C05396=1037.338,216.569,-106.608,170.716,41.966,157.978
C05397=1037.331,216.320,-106.581,170.714,41.965,157.978
C05398=1037.324,216.072,-106.553,170.711,41.964,157.978
C05399=1037.317,215.823,-106.526,170.708,41.963,157.977
C05400=1037.311,215.576,-106.500,170.706,41.962,157.977
C05401=1037.304,215.327,-106.473,170.703,41.961,157.976
C05402=1037.297,215.079,-106.446,170.701,41.960,157.976
C05403=1037.290,214.829,-106.418,170.698,41.959,157.976
C05404=1037.284,214.582,-106.391,170.696,41.958,157.975
C05405=1037.277,214.333,-106.365,170.693,41.957,157.975
C05406=1037.271,214.084,-106.338,170.691,41.956,157.975
C05407=1037.264,213.837,-106.311,170.689,41.955,157.974
C05408=1037.258,213.587,-106.284,170.686,41.953,157.974
C05409=1037.250,213.339,-106.257,170.684,41.953,157.973
C05410=1037.244,213.091,-106.230,170.681,41.952,157.973
C05411=1037.237,212.842,-106.204,170.679,41.951,157.973
C05412=1037.231,212.593,-106.177,170.676,41.950,157.972
C05413=1037.223,212.345,-106.150,170.674,41.949,157.972
C05414=1037.218,212.097,-106.123,170.672,41.947,157.972
C05415=1037.211,211.848,-106.096,170.670,41.946,157.971
C05416=1037.205,211.600,-106.069,170.668,41.945,157.971
C05417=1037.197,211.351,-106.043,170.665,41.944,157.970
C05418=1037.191,211.102,-106.016,170.663,41.943,157.970
C05419=1037.185,210.854,-105.990,170.660,41.942,157.970
C05420=1037.177,210.606,-105.963,170.658,41.941,157.969
C05421=1037.171,210.357,-105.935,170.656,41.940,157.969
C05422=1037.164,210.109,-105.909,170.653,41.939,157.969
C05423=1037.157,209.860,-105.883,170.651,41.938,157.968
C05424=1037.151,209.611,-105.856,170.648,41.937,157.968
C05425=1037.144,209.364,-105.829,170.646,41.936,157.968
C05426=1037.138,209.115,-105.802,170.644,41.935,157.967
C05427=1037.130,208.866,-105.776,170.641,41.934,157.967
C05428=1037.124,208.618,-105.750,170.639,41.933,157.966
C05429=1037.117,208.369,-105.723,170.636,41.932,157.966
C05430=1037.110,208.120,-105.696,170.634,41.931,157.966
C05431=1037.104,207.872,-105.670,170.632,41.930,157.965
C05432=1037.097,207.623,-105.644,170.629,41.928,157.965
C05433=1037.090,207.376,-105.617,170.627,41.927,157.965
C05434=1037.084,207.127,-105.590,170.624,41.926,157.964
C05435=1037.076,206.878,-105.564,170.622,41.925,157.964
C05436=1037.068,206.555,-105.530,170.619,41.924,157.963
C05437=1037.059,206.231,-105.496,170.616,41.923,157.963
C05438=1037.050,205.907,-105.461,170.613,41.921,157.962
C05439=1037.042,205.583,-105.426,170.610,41.921,157.962
C05440=1037.015,204.533,-105.321,170.301,41.816,157.921
C05441=1037.009,204.284,-105.295,170.298,41.816,157.921
C05442=1037.003,204.035,-105.270,170.295,41.816,157.921
C05443=1036.997,203.787,-105.245,170.292,41.815,157.921
C05444=1036.991,203.537,-105.220,170.288,41.815,157.920
C05445=1036.985,203.289,-105.195,170.285,41.815,157.920
C05446=1036.979,203.041,-105.170,170.282,41.814,157.920
C05447=1036.972,202.792,-105.145,170.279,41.814,157.920
C05448=1036.966,202.543,-105.120,170.275,41.814,157.919
C05449=1036.960,202.295,-105.095,170.272,41.813,157.919
C05450=1036.954,202.046,-105.070,170.269,41.813,157.919
C05451=1036.948,201.797,-105.044,170.266,41.813,157.919
C05452=1036.942,201.549,-105.020,170.262,41.813,157.918
C05453=1036.936,201.300,-104.995,170.259,41.813,157.918
C05454=1036.930,201.051,-104.969,170.256,41.812,157.918
C05455=1036.924,200.802,-104.945,170.253,41.812,157.918
C05456=1036.917,200.554,-104.920,170.250,41.812,157.917
C05457=1036.911,200.305,-104.895,170.246,41.812,157.917
C05458=1036.905,200.057,-104.871,170.243,41.812,157.917
C05459=1036.899,199.808,-104.846,170.241,41.811,157.917
C05460=1036.892,199.559,-104.822,170.238,41.811,157.916
C05461=1036.886,199.310,-104.796,170.234,41.811,157.916
C05462=1036.880,199.061,-104.772,170.231,41.811,157.916
C05463=1036.873,198.813,-104.747,170.228,41.811,157.916
C05464=1036.868,198.564,-104.723,170.225,41.811,157.916
C05465=1036.861,198.316,-104.698,170.222,41.811,157.915
C05466=1036.855,198.066,-104.673,170.219,41.810,157.915
C05467=1036.848,197.818,-104.649,170.215,41.810,157.915
C05468=1036.843,197.570,-104.624,170.212,41.810,157.915
C05469=1036.836,197.321,-104.600,170.209,41.810,157.915
C05470=1036.830,197.072,-104.575,170.206,41.810,157.914
C05471=1036.824,196.823,-104.550,170.203,41.810,157.914
C05472=1036.817,196.575,-104.526,170.199,41.810,157.914
C05473=1036.812,196.326,-104.501,170.196,41.810,157.914
C05474=1036.805,196.077,-104.477,170.193,41.809,157.913
C05475=1036.799,195.828,-104.452,170.190,41.810,157.913
C05476=1036.793,195.580,-104.428,170.187,41.810,157.913
C05477=1036.787,195.331,-104.403,170.184,41.809,157.913
C05478=1036.780,195.082,-104.379,170.180,41.809,157.913
C05479=1036.774,194.833,-104.354,170.177,41.809,157.912
C05480=1036.768,194.585,-104.330,170.174,41.809,157.912
C05481=1036.762,194.336,-104.305,170.172,41.809,157.912
C05482=1036.755,194.087,-104.281,170.169,41.809,157.912
C05483=1036.749,193.839,-104.256,170.165,41.809,157.912
C05484=1036.743,193.590,-104.232,170.162,41.808,157.911
C05485=1036.737,193.341,-104.208,170.159,41.809,157.911
C05486=1036.731,193.092,-104.184,170.156,41.809,157.911
C05487=1036.725,192.844,-104.159,170.153,41.808,157.911
C05488=1036.718,192.595,-104.135,170.150,41.808,157.910
C05489=1036.713,192.346,-104.110,170.147,41.809,157.910
C05490=1036.706,192.097,-104.086,170.144,41.808,157.910
C05491=1036.701,191.849,-104.061,170.141,41.808,157.910
C05492=1036.694,191.600,-104.037,170.138,41.808,157.910
C05493=1036.688,191.351,-104.013,170.135,41.808,157.910
C05494=1036.682,191.103,-103.989,170.132,41.808,157.909
C05495=1036.676,190.853,-103.964,170.128,41.808,157.909
C05496=1036.670,190.606,-103.940,170.125,41.808,157.909
C05497=1036.664,190.356,-103.915,170.122,41.808,157.909
C05498=1036.657,190.107,-103.891,170.120,41.808,157.909
C05499=1036.652,189.859,-103.867,170.117,41.807,157.908
C05500=1036.645,189.610,-103.843,170.114,41.807,157.908
C05501=1036.639,189.326,-103.815,170.110,41.807,157.908
C05502=1036.632,189.041,-103.787,170.106,41.808,157.908
C05503=1036.625,188.758,-103.760,170.103,41.807,157.907
C05504=1036.618,188.473,-103.732,170.100,41.807,157.907
C05505=1036.612,188.225,-103.708,170.097,41.807,157.907
C05506=1036.606,187.976,-103.683,170.094,41.807,157.907
C05507=1036.600,187.728,-103.660,170.091,41.807,157.907
C05508=1036.594,187.478,-103.635,170.088,41.807,157.906
C05509=1036.588,187.230,-103.611,170.085,41.807,157.906
C05510=1036.582,186.981,-103.587,170.082,41.807,157.906
C05511=1036.576,186.732,-103.563,170.079,41.807,157.906
C05512=1036.570,186.483,-103.539,170.075,41.807,157.906
C05513=1036.564,186.235,-103.515,170.073,41.807,157.906
C05514=1036.558,185.986,-103.491,170.070,41.807,157.905
C05515=1036.552,185.737,-103.467,170.067,41.806,157.905
C05516=1036.546,185.488,-103.443,170.064,41.806,157.905
C05517=1036.541,185.239,-103.419,170.062,41.806,157.905
C05518=1036.535,184.991,-103.395,170.059,41.806,157.905
C05519=1036.529,184.742,-103.371,170.055,41.806,157.904
C05520=1036.523,184.493,-103.347,170.052,41.806,157.904
C05521=1036.517,184.244,-103.322,170.049,41.806,157.904
C05522=1036.511,183.996,-103.299,170.047,41.806,157.904
C05523=1036.505,183.746,-103.274,170.044,41.806,157.904
C05524=1036.499,183.498,-103.250,170.041,41.806,157.903
C05525=1036.493,183.250,-103.227,170.037,41.806,157.903
C05526=1036.486,183.000,-103.204,170.035,41.806,157.903
C05527=1036.480,182.752,-103.180,170.032,41.807,157.903
C05528=1036.474,182.503,-103.156,170.029,41.806,157.903
C05529=1036.468,182.254,-103.133,170.026,41.807,157.903
C05530=1036.461,182.005,-103.109,170.023,41.807,157.903
C05531=1036.455,181.757,-103.085,170.020,41.807,157.902
C05532=1036.449,181.507,-103.062,170.018,41.807,157.902
C05533=1036.442,181.259,-103.039,170.015,41.807,157.902
C05534=1036.436,181.010,-103.015,170.012,41.807,157.902
C05535=1036.430,180.761,-102.992,170.009,41.808,157.902
C05536=1036.423,180.512,-102.968,170.005,41.808,157.902
C05537=1036.418,180.264,-102.945,170.002,41.808,157.902
C05538=1036.411,180.015,-102.921,170.000,41.808,157.901
C05539=1036.405,179.766,-102.898,169.997,41.808,157.901
C05540=1036.399,179.517,-102.874,169.994,41.809,157.901
C05541=1036.393,179.268,-102.851,169.991,41.809,157.901
C05542=1036.386,179.020,-102.828,169.988,41.809,157.901
C05543=1036.380,178.770,-102.805,169.986,41.809,157.901
C05544=1036.374,178.522,-102.781,169.983,41.810,157.901
C05545=1036.367,178.272,-102.758,169.979,41.809,157.900
C05546=1036.361,178.024,-102.734,169.976,41.810,157.900
C05547=1036.356,177.775,-102.711,169.974,41.810,157.900
C05548=1036.349,177.526,-102.687,169.971,41.810,157.900
C05549=1036.342,177.278,-102.665,169.968,41.810,157.900
C05550=1036.336,177.029,-102.641,169.965,41.811,157.900
C05551=1036.330,176.780,-102.618,169.963,41.810,157.900
C05552=1036.324,176.531,-102.594,169.960,41.811,157.899
C05553=1036.318,176.282,-102.571,169.957,41.811,157.899
C05554=1036.312,176.033,-102.548,169.954,41.811,157.899
C05555=1036.306,175.785,-102.524,169.952,41.811,157.899
C05556=1036.299,175.535,-102.501,169.949,41.812,157.899
C05557=1036.293,175.287,-102.478,169.946,41.812,157.899
C05558=1036.287,175.038,-102.455,169.942,41.812,157.899
C05559=1036.281,174.789,-102.431,169.940,41.812,157.899
C05560=1036.275,174.540,-102.408,169.937,41.813,157.898
C05561=1036.269,174.291,-102.385,169.934,41.812,157.898
C05562=1036.263,174.043,-102.362,169.931,41.813,157.898
C05563=1036.256,173.794,-102.338,169.929,41.813,157.898
C05564=1036.250,173.545,-102.315,169.926,41.813,157.898
C05565=1036.244,173.261,-102.288,169.923,41.813,157.898
C05566=1036.236,172.976,-102.262,169.920,41.814,157.898
C05567=1036.230,172.692,-102.235,169.916,41.813,157.897
C05568=1036.222,172.406,-102.209,169.913,41.814,157.897
C05569=1036.216,172.158,-102.186,169.910,41.814,157.897
C05570=1036.211,171.909,-102.163,169.907,41.814,157.897
C05571=1036.204,171.661,-102.140,169.904,41.814,157.897
C05572=1036.198,171.411,-102.117,169.902,41.815,157.897
C05573=1036.192,171.162,-102.094,169.899,41.815,157.897
C05574=1036.186,170.914,-102.070,169.896,41.815,157.896
C05575=1036.180,170.665,-102.048,169.894,41.815,157.896
C05576=1036.174,170.415,-102.024,169.891,41.816,157.896
C05577=1036.167,170.167,-102.002,169.888,41.816,157.896
C05578=1036.162,169.918,-101.979,169.886,41.816,157.896
C05579=1036.156,169.670,-101.955,169.883,41.816,157.896
C05580=1036.150,169.421,-101.932,169.879,41.817,157.896
C05581=1036.144,169.171,-101.909,169.877,41.816,157.895
C05582=1036.137,168.923,-101.887,169.874,41.817,157.895
C05583=1036.131,168.674,-101.864,169.871,41.817,157.895
C05584=1036.126,168.425,-101.841,169.869,41.817,157.895
C05585=1036.120,168.176,-101.817,169.866,41.817,157.895
C05586=1036.114,167.928,-101.794,169.863,41.818,157.895
C05587=1036.107,167.679,-101.772,169.861,41.818,157.895
C05588=1036.101,167.429,-101.749,169.858,41.818,157.895
C05589=1036.095,167.180,-101.726,169.856,41.818,157.895
C05590=1036.090,166.932,-101.703,169.853,41.818,157.894
C05591=1036.084,166.683,-101.680,169.850,41.819,157.894
C05592=1036.077,166.434,-101.657,169.847,41.818,157.894
C05593=1036.072,166.185,-101.634,169.844,41.819,157.894
C05594=1036.066,165.936,-101.611,169.841,41.819,157.894
C05595=1036.060,165.687,-101.588,169.839,41.819,157.894
C05596=1036.055,165.439,-101.566,169.836,41.819,157.894
C05597=1036.047,165.189,-101.543,169.834,41.820,157.894
C05598=1036.042,164.940,-101.520,169.831,41.820,157.893
C05599=1036.036,164.691,-101.497,169.828,41.820,157.893
C05600=1036.030,164.443,-101.474,169.826,41.820,157.893
C05601=1036.024,164.194,-101.452,169.823,41.820,157.893
C05602=1036.018,163.945,-101.429,169.821,41.821,157.893
C05603=1036.012,163.696,-101.406,169.818,41.821,157.893
C05604=1036.007,163.447,-101.383,169.814,41.821,157.893
C05605=1036.001,163.198,-101.360,169.812,41.821,157.893
C05606=1035.994,162.950,-101.337,169.809,41.822,157.892
C05607=1035.989,162.701,-101.315,169.807,41.822,157.892
C05608=1035.983,162.452,-101.292,169.804,41.822,157.892
C05609=1035.977,162.203,-101.269,169.801,41.822,157.892
C05610=1035.971,161.955,-101.246,169.799,41.822,157.892
C05611=1035.965,161.706,-101.223,169.796,41.823,157.892
C05612=1035.960,161.456,-101.201,169.794,41.822,157.892
C05613=1035.954,161.207,-101.178,169.791,41.823,157.892
C05614=1035.947,160.959,-101.156,169.789,41.823,157.891
C05615=1035.942,160.710,-101.133,169.786,41.824,157.891
C05616=1035.936,160.461,-101.110,169.784,41.823,157.891
C05617=1035.930,160.212,-101.087,169.780,41.824,157.891
C05618=1035.925,159.962,-101.065,169.777,41.824,157.891
C05619=1035.918,159.714,-101.042,169.775,41.824,157.891
C05620=1035.912,159.465,-101.020,169.772,41.825,157.891
C05621=1035.906,159.216,-100.997,169.770,41.825,157.891
C05622=1035.900,158.967,-100.975,169.767,41.825,157.891
C05623=1035.893,158.719,-100.953,169.764,41.826,157.891
C05624=1035.888,158.470,-100.930,169.762,41.826,157.890
C05625=1035.882,158.220,-100.909,169.759,41.827,157.890
C05626=1035.875,157.972,-100.886,169.757,41.827,157.890
C05627=1035.870,157.722,-100.864,169.754,41.827,157.890
C05628=1035.863,157.474,-100.842,169.751,41.828,157.890
C05629=1035.856,157.189,-100.816,169.748,41.828,157.890
C05630=1035.849,156.904,-100.791,169.745,41.829,157.890
C05631=1035.842,156.618,-100.765,169.743,41.829,157.890
C05632=1035.835,156.333,-100.740,169.740,41.829,157.890
C05633=1035.829,156.085,-100.717,169.737,41.830,157.890
C05634=1035.823,155.835,-100.695,169.734,41.830,157.889
C05635=1035.817,155.587,-100.673,169.732,41.830,157.889
C05636=1035.811,155.337,-100.651,169.729,41.831,157.889
C05637=1035.805,155.088,-100.628,169.727,41.831,157.889
C05638=1035.799,154.839,-100.606,169.724,41.831,157.889
C05639=1035.792,154.591,-100.584,169.722,41.832,157.889
C05640=1035.786,154.342,-100.561,169.719,41.832,157.889
C05641=1035.780,154.093,-100.540,169.717,41.832,157.889
C05642=1035.775,153.844,-100.518,169.714,41.833,157.889
C05643=1035.768,153.596,-100.496,169.711,41.833,157.889
C05644=1035.763,153.346,-100.474,169.709,41.834,157.889
C05645=1035.756,153.097,-100.451,169.706,41.834,157.889
C05646=1035.750,152.848,-100.430,169.704,41.834,157.888
C05647=1035.744,152.600,-100.407,169.700,41.835,157.888
C05648=1035.738,152.350,-100.386,169.698,41.835,157.888
C05649=1035.732,152.101,-100.363,169.695,41.835,157.888
C05650=1035.726,151.852,-100.341,169.692,41.836,157.888
C05651=1035.720,151.603,-100.319,169.690,41.836,157.888
C05652=1035.713,151.355,-100.297,169.687,41.837,157.888
C05653=1035.707,151.105,-100.275,169.685,41.837,157.888
C05654=1035.701,150.857,-100.254,169.682,41.837,157.888
C05655=1035.696,150.608,-100.231,169.680,41.838,157.888
C05656=1035.689,150.359,-100.210,169.677,41.839,157.888
C05657=1035.683,150.109,-100.188,169.675,41.839,157.888
C05658=1035.677,149.861,-100.166,169.672,41.839,157.888
C05659=1035.671,149.612,-100.144,169.670,41.840,157.887
C05660=1035.664,149.362,-100.122,169.667,41.840,157.887
C05661=1035.658,149.114,-100.100,169.665,41.840,157.887
C05662=1035.653,148.865,-100.078,169.662,41.841,157.887
C05663=1035.647,148.616,-100.057,169.660,41.841,157.887
C05664=1035.641,148.367,-100.035,169.657,41.841,157.887
C05665=1035.634,148.118,-100.013,169.655,41.842,157.887
C05666=1035.628,147.869,-99.991,169.652,41.842,157.887
C05667=1035.622,147.620,-99.969,169.650,41.842,157.887
C05668=1035.616,147.371,-99.948,169.647,41.843,157.887
C05669=1035.610,147.122,-99.926,169.644,41.844,157.887
C05670=1035.604,146.873,-99.904,169.642,41.844,157.887
C05671=1035.598,146.624,-99.882,169.639,41.845,157.887
C05672=1035.592,146.375,-99.861,169.637,41.845,157.886
C05673=1035.585,146.126,-99.839,169.634,41.845,157.886
C05674=1035.580,145.877,-99.818,169.632,41.846,157.886
C05675=1035.574,145.628,-99.796,169.629,41.847,157.886
C05676=1035.567,145.379,-99.775,169.627,41.847,157.886
C05677=1035.561,145.130,-99.753,169.624,41.847,157.886
C05678=1035.555,144.881,-99.731,169.622,41.848,157.886
C05679=1035.549,144.632,-99.709,169.619,41.848,157.886
C05680=1035.543,144.383,-99.688,169.617,41.849,157.886
C05681=1035.537,144.134,-99.666,169.614,41.849,157.886
C05682=1035.530,143.885,-99.645,169.612,41.850,157.886
C05683=1035.524,143.636,-99.623,169.609,41.850,157.886
C05684=1035.518,143.388,-99.602,169.607,41.850,157.886
C05685=1035.512,143.138,-99.580,169.604,41.851,157.886
C05686=1035.506,142.889,-99.559,169.602,41.852,157.886
C05687=1035.500,142.640,-99.537,169.599,41.852,157.886
C05688=1035.494,142.391,-99.516,169.597,41.852,157.886
C05689=1035.488,142.142,-99.494,169.594,41.853,157.885
C05690=1035.482,141.893,-99.473,169.592,41.853,157.885
C05691=1035.476,141.644,-99.451,169.589,41.854,157.885
C05692=1035.469,141.395,-99.430,169.587,41.854,157.885
C05693=1035.462,141.110,-99.405,169.584,41.855,157.885
C05694=1035.456,140.824,-99.381,169.581,41.855,157.885
C05695=1035.449,140.539,-99.356,169.578,41.856,157.885
C05696=1035.442,140.254,-99.331,169.576,41.857,157.885
C05697=1035.436,140.005,-99.310,169.573,41.857,157.885
C05698=1035.430,139.755,-99.289,169.571,41.857,157.885
C05699=1035.423,139.506,-99.268,169.568,41.858,157.885
C05700=1035.418,139.258,-99.247,169.566,41.858,157.885
C05701=1035.412,139.009,-99.225,169.563,41.859,157.885
C05702=1035.405,138.759,-99.203,169.561,41.859,157.885
C05703=1035.399,138.510,-99.182,169.558,41.860,157.885
C05704=1035.393,138.262,-99.161,169.556,41.860,157.885
C05705=1035.387,138.012,-99.140,169.553,41.861,157.885
C05706=1035.381,137.763,-99.118,169.551,41.861,157.884
C05707=1035.375,137.515,-99.098,169.548,41.862,157.884
C05708=1035.368,137.266,-99.076,169.546,41.862,157.884
C05709=1035.362,137.016,-99.054,169.543,41.863,157.884
C05710=1035.357,136.767,-99.034,169.541,41.864,157.884
C05711=1035.350,136.518,-99.013,169.539,41.864,157.884
C05712=1035.344,136.269,-98.991,169.536,41.865,157.884
C05713=1035.338,136.021,-98.970,169.534,41.865,157.884
C05714=1035.332,135.771,-98.950,169.531,41.866,157.884
C05715=1035.326,135.522,-98.928,169.529,41.866,157.884
C05716=1035.320,135.273,-98.907,169.526,41.867,157.884
C05717=1035.313,135.025,-98.886,169.524,41.867,157.884
C05718=1035.307,134.775,-98.865,169.521,41.868,157.884
C05719=1035.301,134.527,-98.844,169.520,41.869,157.884
C05720=1035.295,134.277,-98.822,169.516,41.869,157.884
C05721=1035.289,134.027,-98.802,169.514,41.869,157.884
C05722=1035.283,133.779,-98.781,169.513,41.870,157.884
C05723=1035.277,133.530,-98.759,169.510,41.871,157.884
C05724=1035.271,133.280,-98.738,169.508,41.871,157.884
C05725=1035.264,133.032,-98.718,169.505,41.871,157.884
C05726=1035.258,132.783,-98.696,169.503,41.872,157.884
C05727=1035.252,132.534,-98.676,169.500,41.873,157.883
C05728=1035.246,132.285,-98.654,169.498,41.873,157.883
C05729=1035.240,132.035,-98.634,169.496,41.874,157.883
C05730=1035.234,131.787,-98.613,169.493,41.874,157.883
C05731=1035.228,131.538,-98.591,169.491,41.875,157.883
C05732=1035.222,131.289,-98.571,169.488,41.875,157.883
C05733=1035.216,131.040,-98.550,169.486,41.876,157.883
C05734=1035.210,130.790,-98.529,169.483,41.876,157.883
C05735=1035.203,130.542,-98.508,169.481,41.877,157.883
C05736=1035.197,130.292,-98.488,169.478,41.878,157.883
C05737=1035.191,130.044,-98.466,169.476,41.878,157.883
C05738=1035.185,129.794,-98.446,169.474,41.879,157.883
C05739=1035.178,129.545,-98.425,169.471,41.879,157.883
C05740=1035.172,129.296,-98.404,169.469,41.880,157.883
C05741=1035.166,129.047,-98.383,169.466,41.881,157.883
C05742=1035.160,128.798,-98.363,169.464,41.882,157.883
C05743=1035.154,128.549,-98.343,169.461,41.882,157.883
C05744=1035.147,128.300,-98.322,169.459,41.882,157.883
C05745=1035.141,128.051,-98.302,169.456,41.883,157.883
C05746=1035.135,127.802,-98.280,169.454,41.884,157.883
C05747=1035.129,127.553,-98.260,169.451,41.885,157.883
C05748=1035.122,127.303,-98.240,169.449,41.885,157.883
C05749=1035.116,127.055,-98.219,169.448,41.886,157.883
C05750=1035.110,126.805,-98.198,169.445,41.886,157.883
C05751=1035.103,126.556,-98.178,169.442,41.887,157.883
C05752=1035.097,126.308,-98.157,169.440,41.888,157.883
C05753=1035.091,126.058,-98.136,169.438,41.888,157.883
C05754=1035.085,125.809,-98.116,169.435,41.889,157.883
C05755=1035.078,125.560,-98.095,169.433,41.889,157.883
C05756=1035.073,125.311,-98.075,169.431,41.890,157.883
C05757=1035.065,125.026,-98.052,169.428,41.891,157.883
C05758=1035.058,124.740,-98.028,169.425,41.892,157.883
C05759=1035.051,124.454,-98.004,169.422,41.892,157.882
C05760=1035.044,124.169,-97.980,169.420,41.893,157.883
C05761=1035.038,123.920,-97.960,169.417,41.894,157.882
C05762=1035.032,123.670,-97.939,169.415,41.894,157.882
C05763=1035.026,123.421,-97.919,169.412,41.895,157.882
C05764=1035.019,123.173,-97.898,169.410,41.895,157.882
C05765=1035.014,122.923,-97.878,169.407,41.896,157.882
C05766=1035.008,122.675,-97.858,169.405,41.897,157.882
C05767=1035.001,122.425,-97.837,169.403,41.897,157.882
C05768=1034.995,122.177,-97.817,169.400,41.898,157.882
C05769=1034.989,121.927,-97.796,169.398,41.898,157.882
C05770=1034.983,121.678,-97.776,169.397,41.899,157.882
C05771=1034.976,121.429,-97.756,169.393,41.900,157.882
C05772=1034.970,121.180,-97.736,169.392,41.900,157.882
C05773=1034.964,120.931,-97.714,169.389,41.901,157.882
C05774=1034.958,120.682,-97.694,169.387,41.901,157.882
C05775=1034.952,120.432,-97.674,169.385,41.902,157.882
C05776=1034.946,120.183,-97.653,169.382,41.903,157.882
C05777=1034.940,119.935,-97.633,169.380,41.903,157.882
C05778=1034.934,119.685,-97.613,169.377,41.904,157.882
C05779=1034.928,119.436,-97.593,169.375,41.904,157.882
C05780=1034.922,119.187,-97.571,169.373,41.905,157.882
C05781=1034.916,118.938,-97.551,169.370,41.906,157.882
C05782=1034.910,118.689,-97.531,169.368,41.906,157.882
C05783=1034.903,118.440,-97.511,169.366,41.907,157.882
C05784=1034.898,118.191,-97.490,169.363,41.907,157.882
C05785=1034.891,117.941,-97.470,169.361,41.908,157.882
C05786=1034.885,117.692,-97.450,169.359,41.908,157.882
C05787=1034.879,117.444,-97.430,169.356,41.909,157.882
C05788=1034.873,117.194,-97.409,169.354,41.910,157.882
C05789=1034.867,116.945,-97.389,169.351,41.910,157.882
C05790=1034.861,116.697,-97.369,169.349,41.911,157.882
C05791=1034.854,116.447,-97.348,169.347,41.911,157.882
C05792=1034.849,116.198,-97.328,169.344,41.912,157.881
C05793=1034.843,115.949,-97.308,169.342,41.913,157.882
C05794=1034.837,115.700,-97.288,169.340,41.913,157.881
C05795=1034.831,115.451,-97.268,169.338,41.914,157.882
C05796=1034.825,115.202,-97.247,169.335,41.914,157.881
C05797=1034.819,114.952,-97.227,169.333,41.915,157.881
C05798=1034.813,114.704,-97.207,169.331,41.916,157.881
C05799=1034.807,114.455,-97.187,169.329,41.916,157.881
C05800=1034.800,114.205,-97.166,169.327,41.916,157.881
C05801=1034.795,113.956,-97.146,169.324,41.917,157.881
C05802=1034.789,113.707,-97.126,169.322,41.918,157.881
C05803=1034.783,113.457,-97.106,169.320,41.918,157.881
C05804=1034.777,113.208,-97.086,169.317,41.919,157.881
C05805=1034.771,112.959,-97.066,169.315,41.919,157.881
C05806=1034.764,112.710,-97.046,169.313,41.920,157.881
C05807=1034.758,112.461,-97.026,169.310,41.921,157.881
C05808=1034.752,112.212,-97.006,169.308,41.922,157.881
C05809=1034.745,111.963,-96.986,169.306,41.922,157.881
C05810=1034.739,111.714,-96.966,169.303,41.923,157.881
C05811=1034.734,111.465,-96.947,169.301,41.923,157.881
C05812=1034.727,111.215,-96.926,169.299,41.924,157.881
C05813=1034.721,110.966,-96.906,169.296,41.925,157.881
C05814=1034.715,110.717,-96.886,169.294,41.925,157.881
C05815=1034.709,110.468,-96.866,169.291,41.926,157.881
C05816=1034.703,110.218,-96.847,169.289,41.927,157.881
C05817=1034.697,109.970,-96.827,169.287,41.927,157.881
C05818=1034.691,109.721,-96.807,169.285,41.928,157.881
C05819=1034.684,109.471,-96.788,169.283,41.929,157.881
C05820=1034.678,109.222,-96.768,169.281,41.929,157.881
C05821=1034.671,108.936,-96.745,169.278,41.930,157.881
C05822=1034.664,108.651,-96.723,169.275,41.931,157.881
C05823=1034.656,108.365,-96.700,169.272,41.932,157.881
C05824=1034.649,108.079,-96.677,169.270,41.933,157.881
C05825=1034.643,107.830,-96.658,169.267,41.933,157.881
C05826=1034.637,107.581,-96.638,169.265,41.934,157.881
C05827=1034.631,107.333,-96.618,169.263,41.935,157.881
C05828=1034.625,107.083,-96.598,169.260,41.936,157.881
C05829=1034.619,106.834,-96.579,169.259,41.937,157.881
C05830=1034.612,106.585,-96.559,169.256,41.937,157.881
C05831=1034.606,106.336,-96.540,169.254,41.938,157.881
C05832=1034.600,106.086,-96.520,169.252,41.938,157.881
C05833=1034.594,105.837,-96.500,169.250,41.939,157.881
C05834=1034.588,105.588,-96.480,169.247,41.940,157.881
C05835=1034.581,105.340,-96.461,169.245,41.941,157.881
C05836=1034.575,105.089,-96.441,169.243,41.941,157.881
C05837=1034.569,104.841,-96.421,169.240,41.942,157.881
C05838=1034.563,104.592,-96.401,169.238,41.942,157.881
C05839=1034.556,104.343,-96.383,169.236,41.943,157.881
C05840=1034.550,104.094,-96.363,169.233,41.944,157.881
C05841=1034.544,103.844,-96.343,169.231,41.944,157.881
C05842=1034.538,103.595,-96.323,169.229,41.945,157.881
C05843=1034.532,103.345,-96.304,169.226,41.946,157.881
C05844=1034.526,103.097,-96.285,169.224,41.947,157.881
C05845=1034.520,102.848,-96.265,169.222,41.947,157.881
C05846=1034.513,102.598,-96.245,169.220,41.948,157.881
C05847=1034.508,102.349,-96.226,169.218,41.948,157.881
C05848=1034.501,102.100,-96.207,169.216,41.949,157.881
C05849=1034.495,101.851,-96.187,169.213,41.950,157.881
C05850=1034.489,101.602,-96.167,169.211,41.951,157.881
C05851=1034.484,101.352,-96.148,169.209,41.951,157.881
C05852=1034.476,101.103,-96.128,169.206,41.952,157.881
C05853=1034.471,100.854,-96.109,169.204,41.952,157.881
C05854=1034.465,100.605,-96.089,169.202,41.953,157.881
C05855=1034.459,100.355,-96.070,169.199,41.954,157.881
C05856=1034.453,100.107,-96.050,169.197,41.955,157.881
C05857=1034.447,99.858,-96.031,169.195,41.955,157.881
C05858=1034.440,99.607,-96.012,169.192,41.956,157.881
C05859=1034.434,99.359,-95.992,169.190,41.957,157.881
C05860=1034.428,99.109,-95.973,169.188,41.957,157.881
C05861=1034.421,98.860,-95.954,169.186,41.958,157.881
C05862=1034.415,98.612,-95.934,169.184,41.959,157.881
C05863=1034.409,98.362,-95.916,169.182,41.959,157.881
C05864=1034.402,98.113,-95.897,169.179,41.961,157.881
C05865=1034.396,97.864,-95.877,169.177,41.961,157.881
C05866=1034.390,97.615,-95.858,169.175,41.962,157.881
C05867=1034.384,97.365,-95.839,169.172,41.963,157.881
C05868=1034.377,97.117,-95.820,169.170,41.963,157.881
C05869=1034.371,96.867,-95.800,169.168,41.964,157.881
C05870=1034.365,96.618,-95.782,169.165,41.965,157.881
C05871=1034.359,96.369,-95.762,169.163,41.965,157.881
C05872=1034.352,96.120,-95.743,169.161,41.966,157.881
C05873=1034.346,95.870,-95.723,169.159,41.967,157.881
C05874=1034.340,95.621,-95.705,169.157,41.968,157.881
C05875=1034.334,95.372,-95.686,169.155,41.969,157.881
C05876=1034.327,95.123,-95.666,169.152,41.969,157.881
C05877=1034.322,94.874,-95.647,169.150,41.970,157.881
C05878=1034.315,94.625,-95.628,169.148,41.971,157.881
C05879=1034.310,94.375,-95.609,169.145,41.971,157.881
C05880=1034.303,94.127,-95.590,169.143,41.972,157.881
C05881=1034.297,93.877,-95.570,169.141,41.973,157.881
C05882=1034.291,93.628,-95.552,169.138,41.974,157.881
C05883=1034.285,93.379,-95.533,169.136,41.975,157.881
C05884=1034.279,93.129,-95.514,169.134,41.975,157.881
C05885=1034.271,92.844,-95.492,169.132,41.976,157.881
C05886=1034.264,92.557,-95.470,169.129,41.977,157.881
C05887=1034.257,92.272,-95.448,169.127,41.977,157.881
C05888=1034.250,91.986,-95.426,169.124,41.978,157.881
C05889=1034.244,91.737,-95.407,169.122,41.979,157.881
C05890=1034.238,91.488,-95.388,169.119,41.980,157.880
C05891=1034.231,91.239,-95.369,169.117,41.981,157.881
C05892=1034.226,90.990,-95.350,169.115,41.981,157.880
C05893=1034.219,90.741,-95.331,169.112,41.982,157.881
C05894=1034.214,90.491,-95.312,169.110,41.982,157.880
C05895=1034.207,90.242,-95.293,169.108,41.983,157.881
C05896=1034.201,89.993,-95.274,169.106,41.984,157.881
C05897=1034.195,89.743,-95.255,169.103,41.985,157.880
C05898=1034.189,89.494,-95.237,169.102,41.986,157.881
C05899=1034.182,89.245,-95.218,169.100,41.987,157.881
C05900=1034.176,88.996,-95.199,169.097,41.987,157.880
C05901=1034.170,88.747,-95.180,169.095,41.988,157.881
C05902=1034.164,88.497,-95.162,169.093,41.989,157.881
C05903=1034.157,88.248,-95.143,169.090,41.990,157.881
C05904=1034.151,87.999,-95.124,169.088,41.990,157.881
C05905=1034.145,87.750,-95.105,169.086,41.991,157.881
C05906=1034.139,87.501,-95.086,169.083,41.992,157.881
C05907=1034.132,87.252,-95.068,169.081,41.993,157.881
C05908=1034.126,87.002,-95.049,169.079,41.993,157.881
C05909=1034.119,86.753,-95.030,169.077,41.995,157.881
C05910=1034.113,86.504,-95.012,169.075,41.995,157.881
C05911=1034.107,86.255,-94.993,169.073,41.996,157.881
C05912=1034.101,86.005,-94.975,169.070,41.997,157.881
C05913=1034.095,85.756,-94.956,169.068,41.998,157.881
C05914=1034.088,85.507,-94.937,169.066,41.998,157.881
C05915=1034.082,85.258,-94.919,169.063,41.999,157.881
C05916=1034.075,85.009,-94.900,169.061,42.000,157.881
C05917=1034.070,84.759,-94.881,169.059,42.000,157.881
C05918=1034.063,84.510,-94.862,169.056,42.001,157.881
C05919=1034.057,84.261,-94.844,169.055,42.002,157.881
C05920=1034.051,84.011,-94.826,169.053,42.003,157.881
C05921=1034.044,83.762,-94.807,169.050,42.004,157.881
C05922=1034.038,83.513,-94.788,169.048,42.005,157.881
C05923=1034.032,83.263,-94.769,169.046,42.005,157.881
C05924=1034.026,83.014,-94.750,169.043,42.006,157.881
C05925=1034.020,82.766,-94.732,169.041,42.007,157.881
C05926=1034.014,82.516,-94.714,169.039,42.007,157.881
C05927=1034.007,82.267,-94.696,169.036,42.008,157.881
C05928=1034.001,82.018,-94.677,169.034,42.009,157.881
C05929=1033.995,81.769,-94.658,169.032,42.010,157.881
C05930=1033.989,81.519,-94.640,169.029,42.011,157.881
C05931=1033.983,81.270,-94.621,169.028,42.012,157.881
C05932=1033.976,81.020,-94.602,169.026,42.012,157.881
C05933=1033.970,80.771,-94.584,169.024,42.013,157.881
C05934=1033.964,80.522,-94.566,169.021,42.014,157.881
C05935=1033.958,80.273,-94.548,169.019,42.014,157.881
C05936=1033.952,80.024,-94.529,169.017,42.015,157.881
C05937=1033.946,79.775,-94.510,169.014,42.016,157.881
C05938=1033.940,79.525,-94.492,169.012,42.017,157.881
C05939=1033.933,79.276,-94.473,169.010,42.017,157.881
C05940=1033.927,79.027,-94.454,169.007,42.018,157.881
C05941=1033.921,78.778,-94.437,169.005,42.019,157.881
C05942=1033.915,78.529,-94.418,169.004,42.020,157.881
C05943=1033.908,78.279,-94.400,169.002,42.020,157.881
C05944=1033.902,78.030,-94.382,168.999,42.021,157.881
C05945=1033.896,77.781,-94.363,168.997,42.022,157.881
C05946=1033.890,77.531,-94.344,168.995,42.022,157.881
C05947=1033.883,77.282,-94.326,168.992,42.023,157.881
C05948=1033.878,77.033,-94.308,168.990,42.024,157.881
C05949=1033.870,76.747,-94.286,168.987,42.025,157.881
C05950=1033.863,76.462,-94.266,168.985,42.026,157.881
C05951=1033.856,76.175,-94.245,168.982,42.027,157.881
C05952=1033.849,75.889,-94.224,168.979,42.028,157.881
C05953=1033.843,75.640,-94.206,168.978,42.029,157.881
C05954=1033.837,75.390,-94.188,168.976,42.030,157.881
C05955=1033.830,75.142,-94.170,168.973,42.030,157.881
C05956=1033.824,74.893,-94.152,168.971,42.031,157.881
C05957=1033.817,74.644,-94.133,168.969,42.032,157.881
C05958=1033.811,74.394,-94.115,168.966,42.033,157.881
C05959=1033.805,74.145,-94.097,168.964,42.033,157.881
C05960=1033.799,73.895,-94.079,168.962,42.034,157.881
C05961=1033.793,73.647,-94.061,168.959,42.036,157.881
C05962=1033.786,73.397,-94.043,168.957,42.036,157.881
C05963=1033.780,73.148,-94.025,168.956,42.037,157.881
C05964=1033.774,72.898,-94.007,168.953,42.038,157.881
C05965=1033.768,72.650,-93.988,168.951,42.039,157.881
C05966=1033.762,72.400,-93.970,168.949,42.039,157.881
C05967=1033.755,72.151,-93.952,168.946,42.040,157.881
C05968=1033.749,71.901,-93.934,168.944,42.041,157.881
C05969=1033.742,71.652,-93.917,168.942,42.041,157.881
C05970=1033.736,71.403,-93.898,168.939,42.042,157.881
C05971=1033.730,71.154,-93.880,168.937,42.043,157.881
C05972=1033.724,70.904,-93.862,168.936,42.044,157.881
C05973=1033.718,70.655,-93.844,168.934,42.045,157.881
C05974=1033.712,70.406,-93.826,168.931,42.046,157.881
C05975=1033.705,70.157,-93.808,168.929,42.047,157.881
C05976=1033.699,69.907,-93.790,168.927,42.047,157.881
C05977=1033.693,69.657,-93.772,168.924,42.048,157.881
C05978=1033.687,69.409,-93.754,168.922,42.049,157.881
C05979=1033.681,69.159,-93.736,168.920,42.050,157.881
C05980=1033.674,68.910,-93.719,168.917,42.050,157.881
C05981=1033.668,68.661,-93.700,168.915,42.051,157.881
C05982=1033.662,68.412,-93.682,168.914,42.052,157.881
C05983=1033.655,68.162,-93.665,168.911,42.053,157.881
C05984=1033.649,67.913,-93.646,168.909,42.054,157.881
C05985=1033.643,67.663,-93.629,168.907,42.055,157.881
C05986=1033.636,67.415,-93.612,168.904,42.056,157.881
C05987=1033.630,67.165,-93.594,168.902,42.057,157.881
C05988=1033.624,66.916,-93.575,168.900,42.057,157.881
C05989=1033.618,66.667,-93.557,168.897,42.058,157.881
C05990=1033.611,66.417,-93.540,168.895,42.059,157.881
C05991=1033.605,66.168,-93.522,168.893,42.060,157.881
C05992=1033.599,65.919,-93.505,168.890,42.060,157.881
C05993=1033.593,65.670,-93.487,168.889,42.061,157.881
C05994=1033.587,65.420,-93.469,168.887,42.062,157.881
C05995=1033.580,65.171,-93.451,168.884,42.063,157.881
C05996=1033.574,64.921,-93.434,168.882,42.064,157.881
C05997=1033.568,64.672,-93.416,168.880,42.064,157.881
C05998=1033.561,64.423,-93.398,168.877,42.066,157.881
C05999=1033.555,64.174,-93.380,168.875,42.067,157.882
C06000=1033.548,63.924,-93.363,168.873,42.067,157.882
C06001=1033.542,63.675,-93.345,168.870,42.068,157.881
C06002=1033.537,63.426,-93.327,168.869,42.069,157.882
C06003=1033.530,63.176,-93.310,168.867,42.070,157.882
C06004=1033.523,62.927,-93.293,168.864,42.071,157.882
C06005=1033.518,62.678,-93.275,168.862,42.072,157.882
C06006=1033.511,62.428,-93.258,168.859,42.073,157.882
C06007=1033.504,62.179,-93.240,168.857,42.074,157.882
C06008=1033.498,61.929,-93.222,168.855,42.075,157.882
C06009=1033.492,61.680,-93.205,168.853,42.076,157.882
C06010=1033.485,61.431,-93.188,168.851,42.076,157.882
C06011=1033.479,61.181,-93.170,168.849,42.077,157.882
C06012=1033.472,60.933,-93.153,168.846,42.078,157.882
C06013=1033.465,60.647,-93.133,168.844,42.079,157.882
C06014=1033.457,60.360,-93.114,168.841,42.080,157.882
C06015=1033.450,60.074,-93.094,168.838,42.081,157.882
C06016=1033.443,59.789,-93.073,168.835,42.082,157.882
C06017=1033.436,59.539,-93.056,168.834,42.083,157.882
C06018=1033.431,59.290,-93.039,168.832,42.084,157.882
C06019=1033.424,59.041,-93.021,168.829,42.085,157.882
C06020=1033.417,58.791,-93.004,168.827,42.086,157.882
C06021=1033.411,58.542,-92.987,168.824,42.087,157.882
C06022=1033.405,58.293,-92.969,168.822,42.088,157.882
C06023=1033.398,58.043,-92.952,168.820,42.089,157.882
C06024=1033.392,57.794,-92.934,168.817,42.090,157.882
C06025=1033.385,57.545,-92.917,168.816,42.091,157.882
C06026=1033.379,57.296,-92.900,168.814,42.092,157.882
C06027=1033.372,57.047,-92.883,168.811,42.093,157.882
C06028=1033.366,56.796,-92.865,168.809,42.094,157.882
C06029=1033.360,56.547,-92.848,168.807,42.095,157.882
C06030=1033.353,56.298,-92.831,168.804,42.095,157.882
C06031=1033.348,56.049,-92.814,168.802,42.096,157.882
C06032=1033.341,55.800,-92.796,168.799,42.097,157.882
C06033=1033.335,55.551,-92.779,168.798,42.098,157.882
C06034=1033.329,55.301,-92.761,168.796,42.099,157.883
C06035=1033.322,55.051,-92.745,168.793,42.100,157.883
C06036=1033.316,54.802,-92.728,168.791,42.100,157.882
C06037=1033.310,54.553,-92.710,168.789,42.101,157.883
C06038=1033.303,54.304,-92.693,168.786,42.102,157.883
C06039=1033.297,54.054,-92.675,168.784,42.103,157.883
C06040=1033.291,53.805,-92.659,168.782,42.104,157.883
C06041=1033.284,53.555,-92.641,168.779,42.105,157.883
C06042=1033.278,53.307,-92.624,168.778,42.106,157.883
C06043=1033.271,53.057,-92.607,168.776,42.107,157.883
C06044=1033.266,52.808,-92.590,168.773,42.108,157.883
C06045=1033.259,52.558,-92.573,168.771,42.109,157.883
C06046=1033.253,52.309,-92.556,168.769,42.110,157.883
C06047=1033.247,52.060,-92.538,168.766,42.110,157.883
C06048=1033.241,51.810,-92.522,168.764,42.111,157.883
C06049=1033.234,51.561,-92.504,168.761,42.112,157.883
C06050=1033.228,51.312,-92.487,168.760,42.113,157.883
C06051=1033.222,51.062,-92.469,168.758,42.113,157.883
C06052=1033.216,50.813,-92.453,168.755,42.114,157.883
C06053=1033.209,50.564,-92.436,168.753,42.115,157.883
C06054=1033.203,50.315,-92.418,168.751,42.116,157.883
C06055=1033.197,50.064,-92.402,168.748,42.117,157.883
C06056=1033.191,49.816,-92.385,168.746,42.118,157.883
C06057=1033.184,49.566,-92.367,168.744,42.119,157.883
C06058=1033.178,49.317,-92.350,168.741,42.120,157.883
C06059=1033.172,49.068,-92.333,168.740,42.121,157.883
C06060=1033.165,48.819,-92.316,168.738,42.121,157.883
C06061=1033.160,48.569,-92.299,168.735,42.122,157.883
C06062=1033.153,48.319,-92.282,168.733,42.123,157.883
C06063=1033.147,48.071,-92.265,168.731,42.124,157.883
C06064=1033.140,47.821,-92.248,168.728,42.124,157.883
C06065=1033.135,47.572,-92.231,168.726,42.125,157.883
C06066=1033.129,47.322,-92.214,168.724,42.126,157.883
C06067=1033.122,47.073,-92.197,168.721,42.127,157.883
C06068=1033.116,46.824,-92.180,168.719,42.128,157.883
C06069=1033.110,46.574,-92.163,168.718,42.129,157.883
C06070=1033.104,46.325,-92.146,168.715,42.130,157.883
C06071=1033.098,46.076,-92.130,168.713,42.131,157.883
C06072=1033.092,45.826,-92.112,168.711,42.131,157.883
C06073=1033.086,45.577,-92.095,168.708,42.132,157.883
C06074=1033.080,45.328,-92.079,168.706,42.133,157.883
C06075=1033.073,45.078,-92.061,168.704,42.134,157.883
C06076=1033.067,44.829,-92.044,168.701,42.134,157.883
C06077=1033.060,44.543,-92.025,168.699,42.135,157.883
C06078=1033.053,44.257,-92.006,168.696,42.136,157.883
C06079=1033.046,43.970,-91.987,168.694,42.137,157.883
C06080=1033.038,43.684,-91.967,168.692,42.138,157.883
C06081=1033.033,43.434,-91.950,168.689,42.139,157.883
C06082=1033.027,43.185,-91.933,168.687,42.140,157.883
C06083=1033.020,42.935,-91.916,168.685,42.141,157.883
C06084=1033.014,42.687,-91.899,168.682,42.142,157.883
C06085=1033.008,42.437,-91.883,168.680,42.142,157.883
C06086=1033.001,42.187,-91.867,168.677,42.143,157.883
C06087=1032.995,41.938,-91.850,168.675,42.144,157.883
C06088=1032.989,41.689,-91.833,168.674,42.145,157.883
C06089=1032.982,41.440,-91.816,168.671,42.146,157.883
C06090=1032.976,41.190,-91.800,168.669,42.147,157.883
C06091=1032.970,40.940,-91.783,168.666,42.148,157.883
C06092=1032.964,40.692,-91.766,168.664,42.149,157.883
C06093=1032.958,40.442,-91.750,168.662,42.150,157.883
C06094=1032.951,40.192,-91.733,168.659,42.151,157.883
C06095=1032.945,39.943,-91.716,168.657,42.152,157.883
C06096=1032.939,39.694,-91.700,168.656,42.152,157.884
C06097=1032.933,39.445,-91.684,168.653,42.154,157.884
C06098=1032.926,39.195,-91.666,168.651,42.154,157.883
C06099=1032.920,38.946,-91.650,168.648,42.155,157.883
C06100=1032.914,38.697,-91.634,168.646,42.156,157.884
C06101=1032.908,38.446,-91.617,168.644,42.157,157.884
C06102=1032.901,38.198,-91.600,168.641,42.158,157.884
C06103=1032.895,37.948,-91.584,168.639,42.158,157.884
C06104=1032.889,37.698,-91.567,168.637,42.159,157.884
C06105=1032.883,37.449,-91.551,168.635,42.160,157.884
C06106=1032.877,37.200,-91.534,168.633,42.161,157.884
C06107=1032.871,36.951,-91.518,168.630,42.162,157.884
C06108=1032.863,36.701,-91.502,168.628,42.163,157.884
C06109=1032.857,36.452,-91.486,168.625,42.164,157.884
C06110=1032.851,36.203,-91.469,168.623,42.165,157.884
C06111=1032.845,35.952,-91.453,168.621,42.166,157.884
C06112=1032.838,35.704,-91.436,168.618,42.167,157.884
C06113=1032.832,35.455,-91.420,168.617,42.168,157.884
C06114=1032.825,35.205,-91.404,168.614,42.169,157.884
C06115=1032.819,34.955,-91.387,168.612,42.170,157.884
C06116=1032.813,34.706,-91.372,168.610,42.171,157.884
C06117=1032.807,34.457,-91.355,168.607,42.172,157.884
C06118=1032.800,34.207,-91.339,168.605,42.173,157.884
C06119=1032.794,33.958,-91.322,168.602,42.174,157.884
C06120=1032.787,33.709,-91.306,168.601,42.175,157.884
C06121=1032.781,33.460,-91.290,168.598,42.176,157.884
C06122=1032.775,33.210,-91.273,168.596,42.177,157.884
C06123=1032.768,32.961,-91.258,168.594,42.178,157.884
C06124=1032.762,32.711,-91.241,168.591,42.178,157.884
C06125=1032.756,32.462,-91.225,168.589,42.179,157.884
C06126=1032.750,32.213,-91.209,168.586,42.180,157.884
C06127=1032.743,31.963,-91.193,168.584,42.181,157.884
C06128=1032.737,31.714,-91.176,168.583,42.182,157.884
C06129=1032.731,31.464,-91.160,168.580,42.183,157.884
C06130=1032.725,31.215,-91.144,168.578,42.184,157.884
C06131=1032.718,30.965,-91.128,168.575,42.185,157.884
C06132=1032.712,30.716,-91.112,168.573,42.186,157.884
C06133=1032.706,30.466,-91.095,168.570,42.187,157.884
C06134=1032.700,30.217,-91.079,168.568,42.188,157.884
C06135=1032.693,29.968,-91.064,168.566,42.189,157.884
C06136=1032.687,29.719,-91.047,168.564,42.190,157.884
C06137=1032.681,29.469,-91.031,168.562,42.191,157.884
C06138=1032.674,29.220,-91.015,168.559,42.192,157.885
C06139=1032.668,28.970,-90.999,168.557,42.193,157.885
C06140=1032.662,28.721,-90.982,168.555,42.193,157.884
C06141=1032.653,28.345,-90.959,168.551,42.195,157.885
C06142=1032.643,27.969,-90.934,168.547,42.196,157.885
C06143=1032.634,27.594,-90.911,168.545,42.198,157.885
C06144=1032.624,27.219,-90.887,168.541,42.199,157.885
C06145=1032.618,26.970,-90.870,168.538,42.200,157.885
C06146=1032.612,26.720,-90.854,168.536,42.201,157.885
C06147=1032.605,26.470,-90.839,168.534,42.202,157.885
C06148=1032.599,26.221,-90.822,168.531,42.203,157.885
C06149=1032.589,25.811,-90.796,168.528,42.205,157.885
C06150=1032.578,25.401,-90.770,168.524,42.206,157.885
C06151=1032.567,24.992,-90.744,168.520,42.208,157.885
C06152=1032.557,24.582,-90.719,168.516,42.210,157.885
C06153=1032.551,24.333,-90.703,168.513,42.211,157.885
C06154=1032.545,24.084,-90.687,168.512,42.212,157.885
C06155=1032.539,23.835,-90.671,168.510,42.213,157.885
C06156=1032.532,23.584,-90.655,168.507,42.214,157.885
C06157=1032.526,23.335,-90.639,168.505,42.215,157.885
C06158=1032.519,23.086,-90.623,168.502,42.216,157.885
C06159=1032.513,22.837,-90.608,168.500,42.217,157.885
C06160=1032.507,22.587,-90.592,168.497,42.218,157.885
C06161=1032.500,22.338,-90.577,168.495,42.218,157.885
C06162=1032.494,22.089,-90.560,168.493,42.219,157.885
C06163=1032.488,21.839,-90.545,168.491,42.220,157.885
C06164=1032.482,21.590,-90.529,168.488,42.221,157.885
C06165=1032.475,21.340,-90.514,168.486,42.222,157.885
C06166=1032.470,21.091,-90.498,168.483,42.223,157.885
C06167=1032.463,20.841,-90.482,168.481,42.224,157.885
C06168=1032.457,20.592,-90.466,168.479,42.225,157.885
C06169=1032.451,20.342,-90.451,168.477,42.226,157.885
C06170=1032.444,20.092,-90.434,168.475,42.227,157.886
C06171=1032.437,19.843,-90.419,168.472,42.228,157.886
C06172=1032.432,19.593,-90.403,168.470,42.229,157.886
C06173=1032.425,19.344,-90.388,168.467,42.230,157.886
C06174=1032.419,19.095,-90.373,168.465,42.231,157.886
C06175=1032.413,18.845,-90.356,168.462,42.232,157.886
C06176=1032.406,18.596,-90.341,168.460,42.233,157.886
C06177=1032.400,18.347,-90.326,168.458,42.234,157.886
C06178=1032.394,18.097,-90.310,168.456,42.235,157.886
C06179=1032.387,17.848,-90.295,168.453,42.236,157.886
C06180=1032.381,17.599,-90.279,168.451,42.237,157.886
C06181=1032.374,17.349,-90.264,168.448,42.238,157.886
C06182=1032.368,17.100,-90.248,168.446,42.239,157.886
C06183=1032.362,16.850,-90.233,168.443,42.240,157.886
C06184=1032.355,16.601,-90.217,168.442,42.241,157.886
C06185=1032.349,16.351,-90.202,168.439,42.242,157.886
C06186=1032.343,16.102,-90.186,168.437,42.243,157.886
C06187=1032.336,15.852,-90.171,168.434,42.244,157.886
C06188=1032.331,15.602,-90.155,168.432,42.245,157.886
C06189=1032.324,15.353,-90.140,168.429,42.246,157.886
C06190=1032.318,15.104,-90.125,168.427,42.247,157.886
C06191=1032.312,14.854,-90.109,168.425,42.248,157.886
C06192=1032.305,14.605,-90.094,168.423,42.249,157.886
C06193=1032.299,14.356,-90.078,168.420,42.250,157.886
C06194=1032.293,14.106,-90.062,168.418,42.251,157.886
C06195=1032.287,13.857,-90.048,168.415,42.252,157.886
C06196=1032.281,13.608,-90.032,168.413,42.253,157.886
C06197=1032.274,13.358,-90.017,168.410,42.254,157.886
C06198=1032.268,13.108,-90.002,168.409,42.255,157.886
C06199=1032.261,12.859,-89.987,168.406,42.257,157.886
C06200=1032.255,12.610,-89.972,168.404,42.257,157.886
C06201=1032.247,12.324,-89.954,168.401,42.259,157.886
C06202=1032.240,12.039,-89.936,168.398,42.260,157.887
C06203=1032.233,11.754,-89.920,168.396,42.261,157.887
C06204=1032.225,11.469,-89.902,168.393,42.263,157.887
C06205=1032.219,11.219,-89.887,168.391,42.264,157.887
C06206=1032.212,10.970,-89.871,168.388,42.265,157.887
C06207=1032.206,10.720,-89.856,168.385,42.266,157.887
C06208=1032.200,10.471,-89.842,168.383,42.267,157.887
C06209=1032.194,10.222,-89.827,168.380,42.268,157.887
C06210=1032.187,9.973,-89.811,168.379,42.269,157.887
C06211=1032.181,9.723,-89.796,168.376,42.271,157.887
C06212=1032.174,9.474,-89.781,168.374,42.272,157.887
C06213=1032.168,9.224,-89.766,168.371,42.273,157.887
C06214=1032.162,8.974,-89.752,168.369,42.274,157.887
C06215=1032.155,8.725,-89.736,168.366,42.275,157.887
C06216=1032.149,8.476,-89.721,168.365,42.276,157.887
C06217=1032.142,8.226,-89.706,168.362,42.277,157.887
C06218=1032.136,7.977,-89.691,168.359,42.278,157.887
C06219=1032.130,7.727,-89.676,168.357,42.279,157.887
C06220=1032.124,7.478,-89.661,168.354,42.280,157.887
C06221=1032.117,7.229,-89.646,168.352,42.281,157.887
C06222=1032.111,6.979,-89.631,168.349,42.282,157.887
C06223=1032.104,6.729,-89.616,168.348,42.283,157.887
C06224=1032.098,6.480,-89.601,168.345,42.284,157.887
C06225=1032.092,6.231,-89.586,168.343,42.285,157.887
C06226=1032.086,5.981,-89.571,168.340,42.286,157.887
C06227=1032.079,5.731,-89.557,168.337,42.287,157.887
C06228=1032.073,5.482,-89.542,168.335,42.288,157.888
C06229=1032.066,5.233,-89.526,168.332,42.289,157.888
C06230=1032.060,4.983,-89.511,168.331,42.290,157.888
C06231=1032.054,4.734,-89.496,168.328,42.291,157.888
C06232=1032.048,4.484,-89.481,168.326,42.292,157.888
C06233=1032.041,4.235,-89.466,168.323,42.293,157.888
C06234=1032.035,3.985,-89.452,168.321,42.294,157.888
C06235=1032.029,3.736,-89.437,168.318,42.295,157.888
C06236=1032.023,3.486,-89.422,168.316,42.296,157.888
C06237=1032.016,3.237,-89.407,168.314,42.298,157.888
C06238=1032.010,2.987,-89.392,168.311,42.299,157.888
C06239=1032.004,2.737,-89.377,168.309,42.300,157.888
C06240=1031.998,2.488,-89.363,168.306,42.301,157.888
C06241=1031.991,2.239,-89.348,168.304,42.302,157.888
C06242=1031.985,1.989,-89.333,168.301,42.303,157.888
C06243=1031.979,1.740,-89.318,168.299,42.304,157.888
C06244=1031.973,1.491,-89.303,168.297,42.305,157.888
C06245=1031.966,1.241,-89.288,168.295,42.306,157.888
C06246=1031.960,0.991,-89.273,168.292,42.307,157.888
C06247=1031.954,0.742,-89.259,168.289,42.308,157.888
C06248=1031.948,0.493,-89.244,168.287,42.309,157.888
C06249=1031.942,0.243,-89.229,168.284,42.310,157.888
C06250=1031.935,-0.007,-89.214,168.282,42.311,157.888
C06251=1031.929,-0.256,-89.199,168.280,42.312,157.888
C06252=1031.923,-0.505,-89.184,168.278,42.313,157.888
C06253=1031.917,-0.756,-89.170,168.275,42.314,157.888
C06254=1031.911,-1.005,-89.156,168.272,42.315,157.888
C06255=1031.905,-1.254,-89.141,168.270,42.316,157.888
C06256=1031.898,-1.504,-89.126,168.267,42.317,157.888
C06257=1031.893,-1.753,-89.111,168.266,42.318,157.888
C06258=1031.886,-2.002,-89.096,168.263,42.319,157.888
C06259=1031.880,-2.252,-89.081,168.261,42.320,157.888
C06260=1031.874,-2.501,-89.067,168.258,42.322,157.888
C06261=1031.868,-2.751,-89.052,168.256,42.323,157.889
C06262=1031.862,-3.001,-89.037,168.253,42.324,157.889
C06263=1031.856,-3.250,-89.023,168.250,42.325,157.889
C06264=1031.849,-3.500,-89.008,168.249,42.326,157.889
C06265=1031.842,-3.783,-88.992,168.246,42.327,157.889
C06266=1031.835,-4.066,-88.974,168.243,42.328,157.889
C06267=1031.828,-4.348,-88.959,168.240,42.329,157.889
C06268=1031.821,-4.632,-88.943,168.237,42.331,157.889
C06269=1031.814,-4.882,-88.928,168.234,42.332,157.889
C06270=1031.808,-5.131,-88.913,168.233,42.333,157.889
C06271=1031.802,-5.380,-88.900,168.230,42.334,157.889
C06272=1031.795,-5.630,-88.885,168.227,42.335,157.889
C06273=1031.788,-5.879,-88.870,168.225,42.336,157.889
C06274=1031.783,-6.129,-88.856,168.222,42.337,157.889
C06275=1031.776,-6.379,-88.841,168.220,42.339,157.889
C06276=1031.769,-6.629,-88.828,168.218,42.340,157.889
C06277=1031.764,-6.878,-88.813,168.215,42.341,157.889
C06278=1031.757,-7.127,-88.798,168.213,42.342,157.889
C06279=1031.751,-7.377,-88.785,168.210,42.343,157.889
C06280=1031.745,-7.626,-88.770,168.207,42.344,157.889
C06281=1031.738,-7.876,-88.756,168.205,42.345,157.889
C06282=1031.732,-8.125,-88.742,168.202,42.346,157.889
C06283=1031.726,-8.375,-88.727,168.200,42.348,157.889
C06284=1031.720,-8.624,-88.714,168.198,42.349,157.889
C06285=1031.713,-8.874,-88.699,168.195,42.350,157.889
C06286=1031.706,-9.124,-88.685,168.192,42.351,157.889
C06287=1031.701,-9.373,-88.670,168.190,42.352,157.889
C06288=1031.694,-9.622,-88.656,168.187,42.353,157.890
C06289=1031.688,-9.871,-88.642,168.186,42.354,157.890
C06290=1031.682,-10.121,-88.627,168.183,42.355,157.890
C06291=1031.676,-10.371,-88.613,168.180,42.357,157.890
C06292=1031.669,-10.620,-88.599,168.178,42.358,157.890
C06293=1031.663,-10.870,-88.585,168.175,42.359,157.890
C06294=1031.656,-11.119,-88.571,168.173,42.360,157.890
C06295=1031.650,-11.369,-88.557,168.171,42.361,157.890
C06296=1031.644,-11.618,-88.542,168.168,42.362,157.890
C06297=1031.638,-11.868,-88.528,168.165,42.364,157.890
C06298=1031.632,-12.117,-88.514,168.163,42.365,157.890
C06299=1031.625,-12.367,-88.500,168.160,42.366,157.890
C06300=1031.620,-12.617,-88.486,168.157,42.367,157.890
C06301=1031.612,-12.866,-88.472,168.156,42.368,157.890
C06302=1031.607,-13.116,-88.458,168.153,42.369,157.890
C06303=1031.601,-13.365,-88.443,168.150,42.371,157.890
C06304=1031.594,-13.615,-88.430,168.148,42.372,157.890
C06305=1031.588,-13.864,-88.415,168.145,42.373,157.890
C06306=1031.582,-14.113,-88.402,168.142,42.374,157.890
C06307=1031.576,-14.364,-88.387,168.141,42.375,157.890
C06308=1031.570,-14.613,-88.373,168.138,42.376,157.890
C06309=1031.563,-14.863,-88.359,168.136,42.377,157.890
C06310=1031.557,-15.112,-88.345,168.133,42.378,157.890
C06311=1031.551,-15.362,-88.331,168.130,42.379,157.890
C06312=1031.545,-15.611,-88.317,168.128,42.380,157.890
C06313=1031.538,-15.860,-88.303,168.125,42.381,157.890
C06314=1031.532,-16.110,-88.289,168.123,42.383,157.891
C06315=1031.526,-16.360,-88.275,168.120,42.384,157.891
C06316=1031.519,-16.609,-88.262,168.118,42.385,157.891
C06317=1031.513,-16.859,-88.247,168.115,42.386,157.891
C06318=1031.507,-17.108,-88.234,168.113,42.388,157.891
C06319=1031.501,-17.357,-88.221,168.111,42.389,157.891
C06320=1031.495,-17.608,-88.206,168.108,42.390,157.891
C06321=1031.488,-17.856,-88.192,168.105,42.391,157.891
C06322=1031.481,-18.106,-88.179,168.102,42.392,157.891
C06323=1031.475,-18.356,-88.165,168.100,42.394,157.891
C06324=1031.469,-18.606,-88.151,168.098,42.395,157.891
C06325=1031.463,-18.855,-88.138,168.095,42.396,157.891
C06326=1031.456,-19.105,-88.124,168.093,42.397,157.891
C06327=1031.450,-19.354,-88.110,168.090,42.398,157.891
C06328=1031.444,-19.603,-88.096,168.087,42.400,157.891
C06329=1031.437,-19.886,-88.081,168.084,42.401,157.891
C06330=1031.430,-20.167,-88.065,168.082,42.402,157.891
C06331=1031.423,-20.448,-88.050,168.079,42.404,157.891
C06332=1031.416,-20.730,-88.035,168.076,42.405,157.891
C06333=1031.409,-20.980,-88.021,168.073,42.406,157.891
C06334=1031.403,-21.229,-88.008,168.070,42.407,157.891
C06335=1031.396,-21.478,-87.993,168.069,42.409,157.892
C06336=1031.391,-21.728,-87.979,168.066,42.410,157.892
C06337=1031.384,-21.977,-87.966,168.063,42.411,157.892
C06338=1031.378,-22.227,-87.953,168.061,42.412,157.892
C06339=1031.372,-22.477,-87.939,168.058,42.413,157.892
C06340=1031.366,-22.726,-87.925,168.055,42.414,157.892
C06341=1031.359,-22.976,-87.912,168.053,42.416,157.892
C06342=1031.354,-23.226,-87.898,168.051,42.417,157.892
C06343=1031.347,-23.475,-87.885,168.048,42.418,157.892
C06344=1031.341,-23.725,-87.871,168.045,42.419,157.892
C06345=1031.334,-23.974,-87.858,168.042,42.421,157.892
C06346=1031.329,-24.224,-87.844,168.040,42.422,157.892
C06347=1031.322,-24.474,-87.830,168.038,42.423,157.892
C06348=1031.316,-24.723,-87.817,168.035,42.424,157.892
C06349=1031.310,-24.972,-87.803,168.033,42.425,157.892
C06350=1031.304,-25.222,-87.789,168.030,42.427,157.892
C06351=1031.297,-25.472,-87.776,168.027,42.428,157.892
C06352=1031.291,-25.721,-87.763,168.024,42.429,157.892
C06353=1031.286,-25.970,-87.749,168.023,42.430,157.892
C06354=1031.279,-26.220,-87.735,168.020,42.432,157.892
C06355=1031.273,-26.470,-87.722,168.017,42.433,157.892
C06356=1031.266,-26.719,-87.709,168.014,42.434,157.892
C06357=1031.261,-26.969,-87.695,168.012,42.435,157.892
C06358=1031.254,-27.218,-87.681,168.009,42.436,157.892
C06359=1031.248,-27.468,-87.668,168.007,42.438,157.892
C06360=1031.242,-27.717,-87.655,168.004,42.439,157.892
C06361=1031.235,-27.967,-87.641,168.002,42.440,157.893
C06362=1031.229,-28.217,-87.629,167.999,42.442,157.893
C06363=1031.223,-28.466,-87.615,167.997,42.443,157.893
C06364=1031.217,-28.715,-87.602,167.994,42.444,157.893
C06365=1031.210,-28.965,-87.589,167.991,42.445,157.893
C06366=1031.203,-29.215,-87.575,167.989,42.447,157.893
C06367=1031.198,-29.465,-87.563,167.986,42.448,157.893
C06368=1031.191,-29.714,-87.549,167.983,42.449,157.893
C06369=1031.185,-29.964,-87.536,167.981,42.451,157.893
C06370=1031.178,-30.213,-87.523,167.978,42.452,157.893
C06371=1031.172,-30.463,-87.510,167.976,42.453,157.893
C06372=1031.166,-30.712,-87.497,167.973,42.454,157.893
C06373=1031.159,-30.962,-87.483,167.970,42.456,157.893
C06374=1031.153,-31.211,-87.470,167.968,42.457,157.893
C06375=1031.147,-31.461,-87.457,167.965,42.458,157.893
C06376=1031.141,-31.711,-87.444,167.963,42.459,157.893
C06377=1031.135,-31.960,-87.431,167.960,42.461,157.893
C06378=1031.129,-32.209,-87.417,167.957,42.462,157.893
C06379=1031.122,-32.460,-87.404,167.955,42.464,157.894
C06380=1031.116,-32.709,-87.391,167.952,42.465,157.894
C06381=1031.110,-32.958,-87.378,167.950,42.466,157.894
C06382=1031.104,-33.208,-87.365,167.947,42.467,157.894
C06383=1031.098,-33.457,-87.352,167.944,42.469,157.894
C06384=1031.091,-33.707,-87.339,167.942,42.470,157.894
C06385=1031.085,-33.957,-87.326,167.939,42.471,157.894
C06386=1031.079,-34.206,-87.313,167.937,42.472,157.894
C06387=1031.072,-34.456,-87.299,167.934,42.474,157.894
C06388=1031.066,-34.706,-87.287,167.931,42.475,157.894
C06389=1031.060,-34.955,-87.274,167.928,42.476,157.894
C06390=1031.054,-35.205,-87.261,167.926,42.478,157.894
C06391=1031.048,-35.454,-87.248,167.924,42.479,157.894
C06392=1031.041,-35.704,-87.234,167.921,42.480,157.894
C06393=1031.035,-35.985,-87.220,167.918,42.481,157.894
C06394=1031.029,-36.266,-87.205,167.915,42.483,157.894
C06395=1031.022,-36.546,-87.191,167.912,42.484,157.894
C06396=1031.014,-36.827,-87.176,167.909,42.486,157.894
C06397=1031.008,-37.076,-87.163,167.906,42.487,157.894
C06398=1031.002,-37.326,-87.150,167.903,42.488,157.894
C06399=1030.996,-37.576,-87.137,167.901,42.489,157.894
C06400=1030.990,-37.825,-87.125,167.899,42.491,157.895
C06401=1030.984,-38.075,-87.111,167.896,42.492,157.895
C06402=1030.977,-38.324,-87.098,167.893,42.493,157.895
C06403=1030.972,-38.574,-87.085,167.890,42.494,157.895
C06404=1030.965,-38.823,-87.072,167.889,42.496,157.895
C06405=1030.959,-39.073,-87.060,167.886,42.497,157.895
C06406=1030.953,-39.323,-87.048,167.883,42.498,157.895
C06407=1030.947,-39.572,-87.034,167.880,42.500,157.895
C06408=1030.941,-39.822,-87.022,167.877,42.501,157.895
C06409=1030.934,-40.071,-87.009,167.875,42.503,157.895
C06410=1030.927,-40.321,-86.996,167.872,42.504,157.895
C06411=1030.921,-40.571,-86.984,167.869,42.505,157.895
C06412=1030.914,-40.820,-86.971,167.867,42.507,157.895
C06413=1030.908,-41.070,-86.958,167.864,42.508,157.895
C06414=1030.903,-41.320,-86.946,167.862,42.509,157.895
C06415=1030.896,-41.569,-86.933,167.859,42.511,157.895
C06416=1030.890,-41.819,-86.921,167.856,42.512,157.895
C06417=1030.884,-42.069,-86.908,167.853,42.514,157.895
C06418=1030.878,-42.318,-86.895,167.850,42.515,157.895
C06419=1030.871,-42.567,-86.883,167.848,42.516,157.896
C06420=1030.865,-42.817,-86.870,167.846,42.517,157.896
C06421=1030.859,-43.067,-86.857,167.843,42.519,157.896
C06422=1030.853,-43.316,-86.845,167.840,42.520,157.896
C06423=1030.846,-43.566,-86.833,167.837,42.521,157.896
C06424=1030.840,-43.816,-86.820,167.835,42.523,157.896
C06425=1030.834,-44.065,-86.807,167.832,42.524,157.896
C06426=1030.827,-44.315,-86.795,167.829,42.526,157.896
C06427=1030.822,-44.565,-86.782,167.826,42.527,157.896
C06428=1030.816,-44.814,-86.770,167.825,42.528,157.896
C06429=1030.809,-45.063,-86.757,167.822,42.530,157.896
C06430=1030.803,-45.313,-86.745,167.819,42.531,157.896
C06431=1030.797,-45.563,-86.732,167.816,42.532,157.896
C06432=1030.791,-45.812,-86.720,167.813,42.534,157.896
C06433=1030.785,-46.062,-86.708,167.811,42.535,157.896
C06434=1030.779,-46.311,-86.694,167.808,42.536,157.896
C06435=1030.772,-46.561,-86.683,167.805,42.538,157.897
C06436=1030.766,-46.811,-86.670,167.802,42.539,157.897
C06437=1030.760,-47.061,-86.657,167.801,42.541,157.897
C06438=1030.754,-47.310,-86.645,167.798,42.542,157.897
C06439=1030.748,-47.560,-86.633,167.795,42.543,157.897
C06440=1030.742,-47.809,-86.621,167.792,42.545,157.897
C06441=1030.735,-48.058,-86.608,167.789,42.546,157.897
C06442=1030.730,-48.308,-86.595,167.786,42.547,157.897
C06443=1030.724,-48.558,-86.583,167.784,42.549,157.897
C06444=1030.717,-48.808,-86.571,167.781,42.550,157.897
C06445=1030.711,-49.057,-86.558,167.778,42.551,157.897
C06446=1030.705,-49.307,-86.546,167.776,42.553,157.897
C06447=1030.699,-49.556,-86.534,167.773,42.554,157.897
C06448=1030.693,-49.806,-86.522,167.771,42.555,157.897
C06449=1030.687,-50.056,-86.509,167.768,42.557,157.897
C06450=1030.681,-50.306,-86.497,167.765,42.558,157.897
C06451=1030.675,-50.555,-86.485,167.762,42.560,157.897
C06452=1030.669,-50.805,-86.472,167.760,42.561,157.897
C06453=1030.662,-51.055,-86.460,167.757,42.563,157.898
C06454=1030.656,-51.304,-86.448,167.754,42.564,157.898
C06455=1030.649,-51.553,-86.437,167.751,42.566,157.898
C06456=1030.644,-51.803,-86.424,167.749,42.568,157.898
C06457=1030.636,-52.085,-86.411,167.746,42.569,157.898
C06458=1030.629,-52.366,-86.397,167.742,42.571,157.898
C06459=1030.622,-52.647,-86.384,167.739,42.573,157.898
C06460=1030.614,-52.928,-86.370,167.737,42.574,157.898
C06461=1030.609,-53.178,-86.359,167.734,42.576,157.898
C06462=1030.603,-53.427,-86.346,167.731,42.577,157.898
C06463=1030.596,-53.677,-86.334,167.729,42.579,157.898
C06464=1030.590,-53.927,-86.322,167.726,42.580,157.898
C06465=1030.583,-54.176,-86.310,167.723,42.582,157.899
C06466=1030.578,-54.425,-86.298,167.720,42.583,157.899
C06467=1030.571,-54.676,-86.287,167.717,42.585,157.899
C06468=1030.565,-54.925,-86.275,167.715,42.587,157.899
C06469=1030.559,-55.175,-86.262,167.712,42.588,157.899
C06470=1030.552,-55.425,-86.250,167.709,42.590,157.899
C06471=1030.546,-55.673,-86.239,167.706,42.591,157.899
C06472=1030.540,-55.924,-86.228,167.704,42.593,157.899
C06473=1030.534,-56.173,-86.215,167.701,42.594,157.899
C06474=1030.527,-56.423,-86.203,167.698,42.596,157.899
C06475=1030.521,-56.672,-86.192,167.695,42.598,157.899
C06476=1030.515,-56.922,-86.180,167.693,42.599,157.899
C06477=1030.509,-57.172,-86.168,167.690,42.600,157.899
C06478=1030.502,-57.422,-86.156,167.687,42.602,157.899
C06479=1030.496,-57.671,-86.145,167.684,42.603,157.900
C06480=1030.490,-57.921,-86.133,167.682,42.605,157.900
C06481=1030.484,-58.171,-86.120,167.679,42.606,157.900
C06482=1030.478,-58.420,-86.109,167.676,42.608,157.900
C06483=1030.471,-58.670,-86.098,167.673,42.609,157.900
C06484=1030.465,-58.919,-86.086,167.671,42.611,157.900
C06485=1030.460,-59.169,-86.074,167.668,42.612,157.900
C06486=1030.453,-59.419,-86.062,167.665,42.614,157.900
C06487=1030.447,-59.668,-86.050,167.662,42.616,157.900
C06488=1030.440,-59.918,-86.039,167.660,42.617,157.900
C06489=1030.435,-60.167,-86.027,167.657,42.619,157.900
C06490=1030.428,-60.417,-86.015,167.654,42.620,157.900
C06491=1030.422,-60.667,-86.004,167.651,42.622,157.901
C06492=1030.416,-60.916,-85.992,167.649,42.624,157.901
C06493=1030.410,-61.167,-85.980,167.646,42.625,157.901
C06494=1030.404,-61.415,-85.969,167.643,42.627,157.901
C06495=1030.398,-61.665,-85.957,167.640,42.628,157.901
C06496=1030.391,-61.915,-85.945,167.638,42.629,157.901
C06497=1030.386,-62.164,-85.933,167.635,42.631,157.901
C06498=1030.380,-62.415,-85.922,167.632,42.632,157.901
C06499=1030.373,-62.664,-85.910,167.629,42.634,157.901
C06500=1030.367,-62.914,-85.899,167.627,42.635,157.901
C06501=1030.361,-63.163,-85.887,167.624,42.637,157.901
C06502=1030.356,-63.413,-85.876,167.621,42.638,157.901
C06503=1030.349,-63.663,-85.864,167.618,42.640,157.901
C06504=1030.343,-63.913,-85.852,167.615,42.641,157.901
C06505=1030.337,-64.162,-85.841,167.613,42.643,157.902
C06506=1030.330,-64.412,-85.830,167.610,42.644,157.902
C06507=1030.325,-64.661,-85.817,167.607,42.646,157.902
C06508=1030.319,-64.911,-85.806,167.605,42.648,157.902
C06509=1030.312,-65.160,-85.795,167.602,42.649,157.902
C06510=1030.306,-65.410,-85.783,167.599,42.651,157.902
C06511=1030.300,-65.659,-85.772,167.596,42.652,157.902
C06512=1030.294,-65.910,-85.760,167.594,42.654,157.902
C06513=1030.289,-66.159,-85.749,167.591,42.655,157.902
C06514=1030.282,-66.409,-85.737,167.588,42.657,157.902
C06515=1030.276,-66.658,-85.726,167.585,42.658,157.902
C06516=1030.270,-66.908,-85.714,167.582,42.660,157.902
C06517=1030.264,-67.158,-85.702,167.580,42.661,157.902
C06518=1030.258,-67.408,-85.691,167.577,42.663,157.902
C06519=1030.252,-67.657,-85.680,167.574,42.664,157.903
C06520=1030.246,-67.907,-85.669,167.571,42.666,157.903
C06521=1030.239,-68.190,-85.656,167.568,42.668,157.903
C06522=1030.232,-68.472,-85.642,167.565,42.669,157.903
C06523=1030.226,-68.754,-85.629,167.561,42.671,157.903
C06524=1030.219,-69.036,-85.617,167.558,42.672,157.903
C06525=1030.213,-69.286,-85.605,167.556,42.674,157.903
C06526=1030.207,-69.536,-85.594,167.553,42.675,157.903
C06527=1030.201,-69.785,-85.583,167.550,42.677,157.903
C06528=1030.195,-70.035,-85.571,167.547,42.678,157.903
C06529=1030.189,-70.284,-85.560,167.545,42.680,157.903
C06530=1030.183,-70.534,-85.548,167.542,42.681,157.903
C06531=1030.177,-70.784,-85.537,167.539,42.683,157.903
C06532=1030.171,-71.034,-85.526,167.536,42.685,157.903
C06533=1030.165,-71.284,-85.515,167.534,42.686,157.903
C06534=1030.159,-71.532,-85.503,167.531,42.688,157.904
C06535=1030.153,-71.783,-85.492,167.528,42.689,157.904
C06536=1030.148,-72.032,-85.481,167.525,42.691,157.904
C06537=1030.142,-72.282,-85.470,167.523,42.692,157.904
///RCONF 1,0,0,1,0,0,0,0,0,0,0,0,0,0,0,0,0,0,0,0,0,0,0,0
C06538=1030.136,-72.532,-85.459,167.520,42.694,157.904
C06539=1030.130,-72.781,-85.447,167.517,42.695,157.904
C06540=1030.124,-73.031,-85.436,167.514,42.697,157.904
C06541=1030.118,-73.281,-85.425,167.511,42.698,157.904
C06542=1030.112,-73.530,-85.414,167.509,42.700,157.904
C06543=1030.106,-73.781,-85.402,167.506,42.701,157.904
C06544=1030.100,-74.029,-85.390,167.503,42.703,157.904
C06545=1030.095,-74.279,-85.380,167.500,42.705,157.904
C06546=1030.088,-74.529,-85.368,167.497,42.706,157.904
C06547=1030.083,-74.779,-85.357,167.494,42.708,157.904
C06548=1030.076,-75.029,-85.347,167.491,42.710,157.904
C06549=1030.070,-75.278,-85.336,167.489,42.711,157.905
C06550=1030.064,-75.527,-85.325,167.486,42.712,157.905
C06551=1030.058,-75.778,-85.314,167.483,42.714,157.905
C06552=1030.052,-76.027,-85.303,167.480,42.716,157.905
C06553=1030.046,-76.277,-85.292,167.478,42.717,157.905
C06554=1030.040,-76.527,-85.281,167.475,42.719,157.905
C06555=1030.033,-76.776,-85.271,167.472,42.721,157.905
C06556=1030.028,-77.026,-85.260,167.469,42.723,157.905
C06557=1030.021,-77.276,-85.248,167.466,42.724,157.905
C06558=1030.016,-77.525,-85.238,167.463,42.726,157.905
C06559=1030.010,-77.775,-85.227,167.460,42.728,157.905
C06560=1030.004,-78.024,-85.216,167.458,42.730,157.906
C06561=1029.998,-78.274,-85.205,167.455,42.731,157.906
C06562=1029.992,-78.524,-85.194,167.452,42.732,157.906
C06563=1029.986,-78.773,-85.183,167.449,42.734,157.906
C06564=1029.979,-79.023,-85.172,167.447,42.735,157.906
C06565=1029.974,-79.273,-85.162,167.444,42.737,157.906
C06566=1029.968,-79.523,-85.151,167.440,42.739,157.906
C06567=1029.962,-79.773,-85.140,167.438,42.741,157.906
C06568=1029.956,-80.023,-85.129,167.435,42.742,157.906
C06569=1029.949,-80.272,-85.119,167.432,42.744,157.906
C06570=1029.944,-80.521,-85.108,167.429,42.746,157.906
C06571=1029.937,-80.772,-85.098,167.427,42.748,157.906
C06572=1029.931,-81.021,-85.087,167.424,42.750,157.907
C06573=1029.925,-81.271,-85.076,167.420,42.752,157.907
C06574=1029.919,-81.520,-85.066,167.418,42.753,157.907
C06575=1029.913,-81.771,-85.055,167.415,42.755,157.907
C06576=1029.906,-82.020,-85.045,167.412,42.757,157.907
C06577=1029.901,-82.269,-85.034,167.409,42.758,157.907
C06578=1029.895,-82.519,-85.023,167.407,42.760,157.907
C06579=1029.888,-82.769,-85.013,167.404,42.762,157.907
C06580=1029.882,-83.019,-85.002,167.400,42.764,157.907
C06581=1029.876,-83.268,-84.992,167.398,42.766,157.908
C06582=1029.871,-83.518,-84.982,167.395,42.767,157.908
C06583=1029.864,-83.768,-84.971,167.392,42.769,157.908
C06584=1029.858,-84.017,-84.961,167.390,42.771,157.908
C06585=1029.851,-84.302,-84.949,167.386,42.773,157.908
C06586=1029.844,-84.587,-84.937,167.383,42.775,157.908
C06587=1029.838,-84.871,-84.925,167.380,42.777,157.908
C06588=1029.830,-85.156,-84.913,167.376,42.779,157.908
C06589=1029.824,-85.405,-84.903,167.373,42.781,157.908
C06590=1029.819,-85.655,-84.892,167.371,42.783,157.908
C06591=1029.812,-85.904,-84.882,167.368,42.784,157.909
C06592=1029.807,-86.154,-84.871,167.365,42.786,157.909
C06593=1029.801,-86.404,-84.862,167.362,42.788,157.909
C06594=1029.794,-86.654,-84.850,167.359,42.790,157.909
C06595=1029.788,-86.904,-84.841,167.356,42.792,157.909
C06596=1029.782,-87.153,-84.830,167.353,42.793,157.909
C06597=1029.777,-87.403,-84.819,167.351,42.795,157.909
C06598=1029.770,-87.653,-84.809,167.348,42.797,157.909
C06599=1029.765,-87.902,-84.799,167.345,42.799,157.909
C06600=1029.758,-88.152,-84.789,167.342,42.800,157.909
C06601=1029.753,-88.401,-84.778,167.339,42.802,157.910
C06602=1029.746,-88.652,-84.768,167.336,42.804,157.910
C06603=1029.740,-88.901,-84.757,167.334,42.806,157.910
C06604=1029.734,-89.151,-84.748,167.331,42.808,157.910
C06605=1029.728,-89.401,-84.737,167.328,42.810,157.910
C06606=1029.722,-89.650,-84.727,167.324,42.811,157.910
C06607=1029.716,-89.900,-84.716,167.322,42.813,157.910
C06608=1029.711,-90.150,-84.706,167.319,42.815,157.910
C06609=1029.704,-90.399,-84.696,167.316,42.816,157.910
C06610=1029.699,-90.649,-84.686,167.314,42.818,157.911
C06611=1029.693,-90.898,-84.676,167.310,42.820,157.911
C06612=1029.687,-91.149,-84.665,167.307,42.822,157.911
C06613=1029.681,-91.398,-84.656,167.305,42.824,157.911
C06614=1029.675,-91.648,-84.645,167.302,42.826,157.911
C06615=1029.669,-91.898,-84.635,167.299,42.827,157.911
C06616=1029.663,-92.147,-84.625,167.297,42.829,157.911
C06617=1029.657,-92.397,-84.615,167.293,42.831,157.911
C06618=1029.652,-92.647,-84.605,167.290,42.833,157.911
C06619=1029.645,-92.896,-84.595,167.287,42.834,157.911
C06620=1029.640,-93.146,-84.584,167.285,42.836,157.912
C06621=1029.633,-93.396,-84.574,167.282,42.838,157.912
C06622=1029.628,-93.646,-84.564,167.279,42.840,157.912
C06623=1029.622,-93.895,-84.554,167.276,42.842,157.912
C06624=1029.616,-94.145,-84.543,167.273,42.843,157.912
C06625=1029.610,-94.395,-84.534,167.270,42.845,157.912
C06626=1029.604,-94.645,-84.524,167.268,42.847,157.912
C06627=1029.599,-94.894,-84.513,167.265,42.849,157.912
C06628=1029.592,-95.144,-84.503,167.262,42.850,157.912
C06629=1029.587,-95.394,-84.493,167.259,42.852,157.912
C06630=1029.581,-95.644,-84.484,167.256,42.854,157.912
C06631=1029.575,-95.894,-84.473,167.253,42.856,157.913
C06632=1029.570,-96.143,-84.463,167.251,42.858,157.913
C06633=1029.564,-96.393,-84.453,167.248,42.859,157.913
///RCONF 1,0,0,0,0,0,0,0,0,0,0,0,0,0,0,0,0,0,0,0,0,0,0,0
C06634=1029.558,-96.643,-84.444,167.245,42.861,157.913
C06635=1029.551,-96.892,-84.433,167.241,42.863,157.913
C06636=1029.546,-97.142,-84.423,167.239,42.865,157.913
C06637=1029.540,-97.392,-84.414,167.236,42.867,157.913
C06638=1029.534,-97.642,-84.404,167.233,42.868,157.913
C06639=1029.528,-97.892,-84.394,167.231,42.870,157.913
C06640=1029.522,-98.141,-84.384,167.227,42.872,157.913
C06641=1029.516,-98.391,-84.374,167.224,42.874,157.914
C06642=1029.511,-98.640,-84.364,167.222,42.876,157.914
C06643=1029.505,-98.890,-84.355,167.219,42.878,157.914
C06644=1029.498,-99.139,-84.345,167.215,42.880,157.914
C06645=1029.493,-99.390,-84.335,167.213,42.882,157.914
C06646=1029.487,-99.639,-84.326,167.210,42.884,157.914
C06647=1029.481,-99.889,-84.316,167.207,42.886,157.914
C06648=1029.474,-100.139,-84.306,167.205,42.888,157.914
C06649=1029.468,-100.426,-84.295,167.201,42.890,157.915
C06650=1029.462,-100.712,-84.283,167.197,42.892,157.915
C06651=1029.455,-100.999,-84.272,167.194,42.895,157.915
C06652=1029.447,-101.286,-84.261,167.191,42.896,157.915
C06653=1029.442,-101.535,-84.252,167.187,42.898,157.915
C06654=1029.436,-101.785,-84.242,167.185,42.900,157.915
C06655=1029.430,-102.035,-84.233,167.182,42.902,157.915
C06656=1029.424,-102.285,-84.223,167.179,42.904,157.915
C06657=1029.418,-102.534,-84.213,167.177,42.906,157.915
C06658=1029.412,-102.784,-84.204,167.173,42.908,157.916
C06659=1029.406,-103.033,-84.194,167.171,42.910,157.916
C06660=1029.401,-103.283,-84.184,167.168,42.912,157.916
C06661=1029.395,-103.533,-84.175,167.165,42.914,157.916
C06662=1029.389,-103.784,-84.166,167.162,42.916,157.916
C06663=1029.383,-104.033,-84.157,167.159,42.918,157.916
C06664=1029.377,-104.283,-84.147,167.156,42.920,157.916
C06665=1029.371,-104.532,-84.137,167.154,42.922,157.916
C06666=1029.365,-104.782,-84.127,167.150,42.924,157.917
C06667=1029.360,-105.032,-84.118,167.147,42.925,157.917
C06668=1029.354,-105.281,-84.109,167.145,42.927,157.917
C06669=1029.347,-105.531,-84.099,167.142,42.930,157.917
C06670=1029.341,-105.781,-84.089,167.138,42.932,157.917
C06671=1029.336,-106.031,-84.081,167.136,42.934,157.917
C06672=1029.331,-106.281,-84.071,167.133,42.935,157.917
C06673=1029.324,-106.531,-84.061,167.130,42.937,157.917
C06674=1029.319,-106.780,-84.052,167.127,42.939,157.917
C06675=1029.313,-107.029,-84.042,167.124,42.941,157.918
C06676=1029.307,-107.280,-84.034,167.121,42.943,157.918
C06677=1029.301,-107.530,-84.024,167.119,42.945,157.918
C06678=1029.295,-107.779,-84.015,167.115,42.948,157.918
C06679=1029.289,-108.029,-84.005,167.113,42.949,157.918
C06680=1029.283,-108.279,-83.996,167.110,42.951,157.918
C06681=1029.277,-108.528,-83.987,167.107,42.953,157.918
C06682=1029.271,-108.778,-83.978,167.103,42.955,157.918
C06683=1029.265,-109.028,-83.968,167.101,42.958,157.919
C06684=1029.260,-109.277,-83.960,167.098,42.959,157.919
C06685=1029.254,-109.527,-83.950,167.095,42.961,157.919
C06686=1029.248,-109.777,-83.940,167.092,42.963,157.919
C06687=1029.242,-110.027,-83.932,167.090,42.966,157.919
C06688=1029.236,-110.276,-83.922,167.087,42.968,157.919
C06689=1029.230,-110.526,-83.913,167.083,42.970,157.919
C06690=1029.225,-110.776,-83.904,167.080,42.972,157.920
C06691=1029.219,-111.026,-83.895,167.078,42.973,157.920
C06692=1029.212,-111.276,-83.885,167.075,42.976,157.920
C06693=1029.207,-111.525,-83.877,167.072,42.978,157.920
C06694=1029.201,-111.775,-83.867,167.069,42.980,157.920
C06695=1029.196,-112.025,-83.859,167.066,42.982,157.920
C06696=1029.189,-112.275,-83.849,167.063,42.984,157.920
C06697=1029.183,-112.524,-83.840,167.060,42.986,157.921
C06698=1029.178,-112.774,-83.831,167.057,42.988,157.921
C06699=1029.172,-113.024,-83.821,167.055,42.990,157.921
C06700=1029.167,-113.274,-83.813,167.051,42.992,157.921
C06701=1029.160,-113.523,-83.803,167.048,42.994,157.921
C06702=1029.155,-113.773,-83.795,167.046,42.996,157.921
C06703=1029.149,-114.023,-83.785,167.042,42.998,157.921
C06704=1029.143,-114.273,-83.777,167.040,43.000,157.921
C06705=1029.138,-114.522,-83.767,167.037,43.002,157.921
C06706=1029.132,-114.773,-83.758,167.034,43.005,157.922
C06707=1029.125,-115.022,-83.750,167.031,43.007,157.922
C06708=1029.120,-115.272,-83.741,167.028,43.008,157.922
C06709=1029.114,-115.521,-83.732,167.026,43.011,157.922
C06710=1029.108,-115.772,-83.723,167.022,43.013,157.922
C06711=1029.102,-116.021,-83.714,167.019,43.015,157.922
C06712=1029.097,-116.271,-83.705,167.017,43.017,157.922
C06713=1029.090,-116.557,-83.695,167.013,43.019,157.923
C06714=1029.083,-116.843,-83.684,167.010,43.022,157.923
C06715=1029.077,-117.130,-83.675,167.006,43.024,157.923
C06716=1029.070,-117.416,-83.664,167.003,43.027,157.923
C06717=1029.065,-117.666,-83.656,167.000,43.029,157.923
C06718=1029.058,-117.915,-83.647,166.997,43.031,157.923
C06719=1029.052,-118.165,-83.638,166.995,43.033,157.924
C06720=1029.047,-118.415,-83.629,166.991,43.035,157.924
C06721=1029.041,-118.665,-83.620,166.988,43.038,157.924
C06722=1029.035,-118.915,-83.611,166.986,43.040,157.924
C06723=1029.029,-119.164,-83.603,166.983,43.041,157.924
C06724=1029.024,-119.413,-83.594,166.980,43.044,157.924
C06725=1029.018,-119.664,-83.585,166.977,43.046,157.924
C06726=1029.012,-119.914,-83.577,166.974,43.048,157.924
C06727=1029.006,-120.164,-83.569,166.971,43.051,157.925
C06728=1029.000,-120.413,-83.559,166.968,43.052,157.925
C06729=1028.994,-120.663,-83.550,166.965,43.054,157.925
C06730=1028.989,-120.913,-83.542,166.962,43.057,157.925
C06731=1028.984,-121.163,-83.534,166.959,43.059,157.925
C06732=1028.977,-121.412,-83.525,166.957,43.061,157.925
C06733=1028.972,-121.662,-83.516,166.953,43.063,157.925
C06734=1028.966,-121.912,-83.507,166.950,43.065,157.926
C06735=1028.960,-122.162,-83.499,166.948,43.067,157.926
C06736=1028.954,-122.411,-83.490,166.944,43.070,157.926
C06737=1028.948,-122.661,-83.481,166.942,43.072,157.926
C06738=1028.943,-122.911,-83.473,166.939,43.074,157.926
C06739=1028.936,-123.161,-83.465,166.937,43.076,157.926
C06740=1028.931,-123.411,-83.456,166.933,43.078,157.926
C06741=1028.926,-123.660,-83.448,166.930,43.081,157.927
C06742=1028.920,-123.910,-83.438,166.928,43.083,157.927
C06743=1028.914,-124.160,-83.430,166.924,43.085,157.927
C06744=1028.908,-124.409,-83.422,166.922,43.087,157.927
C06745=1028.903,-124.660,-83.413,166.919,43.089,157.927
C06746=1028.897,-124.909,-83.405,166.915,43.092,157.927
C06747=1028.891,-125.159,-83.396,166.913,43.094,157.927
C06748=1028.885,-125.409,-83.388,166.910,43.096,157.928
C06749=1028.879,-125.659,-83.380,166.907,43.098,157.928
C06750=1028.874,-125.908,-83.371,166.904,43.101,157.928
C06751=1028.868,-126.159,-83.363,166.901,43.103,157.928
C06752=1028.862,-126.408,-83.354,166.898,43.105,157.928
C06753=1028.856,-126.658,-83.347,166.895,43.107,157.928
C06754=1028.850,-126.908,-83.338,166.893,43.109,157.929
C06755=1028.844,-127.157,-83.330,166.889,43.112,157.929
C06756=1028.839,-127.407,-83.321,166.886,43.114,157.929
C06757=1028.833,-127.657,-83.313,166.884,43.116,157.929
C06758=1028.828,-127.906,-83.304,166.880,43.118,157.929
C06759=1028.822,-128.155,-83.296,166.878,43.120,157.929
C06760=1028.818,-128.405,-83.287,166.875,43.121,157.929
C06761=1028.814,-128.655,-83.276,166.872,43.122,157.929
C06762=1028.810,-128.905,-83.265,166.870,43.123,157.929
C06763=1028.808,-129.155,-83.255,166.868,43.122,157.929
C06764=1028.805,-129.404,-83.242,166.865,43.122,157.929
C06765=1028.803,-129.654,-83.231,166.863,43.121,157.928
C06766=1028.803,-129.904,-83.217,166.860,43.120,157.928
C06767=1028.802,-130.154,-83.204,166.859,43.118,157.927
C06768=1028.802,-130.404,-83.190,166.856,43.115,157.927
C06769=1028.803,-130.654,-83.176,166.854,43.112,157.926
C06770=1028.805,-130.903,-83.160,166.852,43.109,157.925
C06771=1028.806,-131.154,-83.144,166.851,43.105,157.925
C06772=1028.810,-131.403,-83.128,166.849,43.101,157.924
C06773=1028.813,-131.653,-83.111,166.847,43.097,157.923
C06774=1028.816,-131.903,-83.094,166.846,43.091,157.922
C06775=1028.821,-132.153,-83.075,166.845,43.085,157.921
C06776=1028.826,-132.402,-83.057,166.844,43.079,157.920
C06777=1028.512,-132.428,-83.367,166.794,43.328,157.958
C06778=1028.506,-132.178,-83.385,166.796,43.334,157.959
C06779=1028.502,-131.928,-83.404,166.798,43.340,157.960
C06780=1028.498,-131.679,-83.421,166.799,43.344,157.961
C06781=1028.496,-131.428,-83.438,166.801,43.349,157.962
C06782=1028.492,-131.178,-83.455,166.802,43.353,157.962
C06783=1028.490,-130.929,-83.470,166.804,43.357,157.963
C06784=1028.489,-130.679,-83.486,166.806,43.361,157.964
C06785=1028.488,-130.429,-83.500,166.808,43.363,157.965
C06786=1028.488,-130.179,-83.514,166.810,43.366,157.965
C06787=1028.488,-129.929,-83.527,166.812,43.368,157.966
C06788=1028.489,-129.679,-83.541,166.814,43.370,157.966
C06789=1028.491,-129.430,-83.553,166.817,43.371,157.966
C06790=1028.493,-129.180,-83.565,166.819,43.371,157.967
C06791=1028.496,-128.930,-83.576,166.821,43.371,157.967
C06792=1028.499,-128.681,-83.586,166.824,43.371,157.967
C06793=1028.503,-128.431,-83.597,166.826,43.370,157.967
C06794=1028.508,-128.181,-83.606,166.829,43.369,157.967
C06795=1028.513,-127.932,-83.616,166.832,43.367,157.967
C06796=1028.519,-127.682,-83.623,166.835,43.364,157.967
C06797=1028.524,-127.432,-83.632,166.838,43.362,157.967
C06798=1028.530,-127.183,-83.640,166.841,43.359,157.967
C06799=1028.536,-126.933,-83.649,166.844,43.358,157.966
C06800=1028.542,-126.683,-83.657,166.846,43.355,157.966
C06801=1028.547,-126.433,-83.665,166.850,43.353,157.966
C06802=1028.554,-126.183,-83.673,166.852,43.350,157.966
C06803=1028.559,-125.934,-83.682,166.855,43.348,157.966
C06804=1028.564,-125.684,-83.690,166.859,43.346,157.966
C06805=1028.570,-125.435,-83.698,166.861,43.344,157.966
C06806=1028.576,-125.184,-83.707,166.864,43.341,157.965
C06807=1028.582,-124.935,-83.715,166.867,43.339,157.965
C06808=1028.587,-124.685,-83.723,166.870,43.337,157.965
C06809=1028.593,-124.435,-83.732,166.874,43.335,157.965
C06810=1028.599,-124.185,-83.740,166.876,43.333,157.965
C06811=1028.605,-123.936,-83.749,166.879,43.330,157.965
C06812=1028.611,-123.686,-83.758,166.882,43.328,157.965
C06813=1028.617,-123.436,-83.766,166.885,43.326,157.964
C06814=1028.622,-123.187,-83.775,166.887,43.324,157.964
C06815=1028.628,-122.936,-83.783,166.891,43.322,157.964
C06816=1028.633,-122.686,-83.792,166.894,43.319,157.964
C06817=1028.640,-122.436,-83.800,166.896,43.317,157.964
C06818=1028.645,-122.187,-83.809,166.900,43.314,157.964
C06819=1028.650,-121.938,-83.818,166.902,43.313,157.963
C06820=1028.657,-121.687,-83.826,166.905,43.311,157.963
C06821=1028.662,-121.438,-83.835,166.908,43.308,157.963
C06822=1028.667,-121.188,-83.843,166.911,43.306,157.963
C06823=1028.674,-120.938,-83.853,166.914,43.303,157.963
C06824=1028.680,-120.689,-83.861,166.917,43.301,157.963
C06825=1028.686,-120.438,-83.869,166.920,43.300,157.963
C06826=1028.691,-120.189,-83.878,166.922,43.297,157.962
C06827=1028.697,-119.939,-83.887,166.926,43.295,157.962
C06828=1028.702,-119.689,-83.896,166.929,43.292,157.962
C06829=1028.708,-119.440,-83.904,166.931,43.290,157.962
C06830=1028.714,-119.189,-83.913,166.935,43.288,157.962
C06831=1028.720,-118.940,-83.922,166.937,43.286,157.962
C06832=1028.726,-118.690,-83.931,166.940,43.284,157.962
C06833=1028.732,-118.440,-83.939,166.944,43.282,157.962
C06834=1028.738,-118.191,-83.948,166.946,43.279,157.961
C06835=1028.743,-117.941,-83.957,166.949,43.278,157.961
C06836=1028.749,-117.690,-83.966,166.952,43.275,157.961
C06837=1028.754,-117.441,-83.975,166.955,43.273,157.961
C06838=1028.762,-117.154,-83.984,166.958,43.270,157.961
C06839=1028.768,-116.869,-83.995,166.962,43.268,157.961
C06840=1028.775,-116.583,-84.005,166.965,43.266,157.960
C06841=1028.781,-116.296,-84.015,166.968,43.263,157.960
C06842=1028.787,-116.047,-84.023,166.972,43.261,157.960
C06843=1028.793,-115.797,-84.032,166.974,43.259,157.960
C06844=1028.799,-115.547,-84.042,166.977,43.256,157.960
C06845=1028.805,-115.297,-84.050,166.980,43.254,157.960
C06846=1028.810,-115.048,-84.060,166.983,43.252,157.960
C06847=1028.816,-114.797,-84.068,166.986,43.250,157.959
C06848=1028.822,-114.548,-84.078,166.988,43.248,157.959
C06849=1028.828,-114.298,-84.086,166.992,43.246,157.959
C06850=1028.834,-114.049,-84.095,166.994,43.243,157.959
C06851=1028.840,-113.799,-84.104,166.997,43.242,157.959
C06852=1028.846,-113.549,-84.113,167.001,43.240,157.959
C06853=1028.851,-113.299,-84.122,167.003,43.238,157.959
C06854=1028.857,-113.049,-84.132,167.006,43.235,157.959
C06855=1028.862,-112.800,-84.140,167.010,43.233,157.958
C06856=1028.869,-112.550,-84.150,167.012,43.231,157.958
C06857=1028.874,-112.300,-84.158,167.015,43.229,157.958
C06858=1028.880,-112.050,-84.168,167.018,43.227,157.958
C06859=1028.886,-111.800,-84.176,167.021,43.225,157.958
C06860=1028.891,-111.551,-84.186,167.024,43.223,157.958
C06861=1028.898,-111.301,-84.195,167.026,43.221,157.958
C06862=1028.903,-111.051,-84.204,167.030,43.218,157.958
C06863=1028.909,-110.802,-84.213,167.033,43.216,157.957
C06864=1028.915,-110.552,-84.223,167.035,43.214,157.957
C06865=1028.921,-110.302,-84.231,167.039,43.212,157.957
C06866=1028.927,-110.052,-84.241,167.041,43.210,157.957
C06867=1028.933,-109.802,-84.250,167.044,43.208,157.957
C06868=1028.938,-109.553,-84.259,167.048,43.206,157.957
C06869=1028.944,-109.303,-84.269,167.050,43.203,157.957
C06870=1028.950,-109.053,-84.277,167.053,43.202,157.956
C06871=1028.956,-108.803,-84.287,167.055,43.200,157.956
C06872=1028.962,-108.554,-84.296,167.059,43.198,157.956
C06873=1028.968,-108.304,-84.306,167.062,43.195,157.956
C06874=1028.973,-108.054,-84.314,167.064,43.193,157.956
C06875=1028.980,-107.804,-84.324,167.068,43.191,157.956
C06876=1028.986,-107.555,-84.333,167.071,43.189,157.956
C06877=1028.991,-107.305,-84.342,167.073,43.187,157.956
C06878=1028.997,-107.055,-84.351,167.077,43.185,157.955
C06879=1029.003,-106.805,-84.361,167.079,43.183,157.955
C06880=1029.008,-106.556,-84.371,167.082,43.181,157.955
C06881=1029.014,-106.306,-84.380,167.085,43.179,157.955
C06882=1029.020,-106.056,-84.389,167.088,43.177,157.955
C06883=1029.026,-105.806,-84.399,167.091,43.175,157.955
C06884=1029.032,-105.557,-84.408,167.094,43.173,157.955
C06885=1029.038,-105.307,-84.418,167.096,43.171,157.955
C06886=1029.044,-105.057,-84.427,167.100,43.169,157.955
C06887=1029.049,-104.808,-84.437,167.103,43.167,157.954
C06888=1029.055,-104.558,-84.446,167.105,43.165,157.954
C06889=1029.061,-104.308,-84.455,167.109,43.163,157.954
C06890=1029.067,-104.058,-84.465,167.111,43.161,157.954
C06891=1029.073,-103.809,-84.474,167.114,43.159,157.954
C06892=1029.079,-103.559,-84.484,167.117,43.157,157.954
C06893=1029.084,-103.309,-84.494,167.120,43.155,157.954
C06894=1029.091,-103.059,-84.503,167.123,43.153,157.954
C06895=1029.096,-102.810,-84.513,167.126,43.151,157.953
C06896=1029.102,-102.560,-84.522,167.128,43.149,157.953
C06897=1029.108,-102.310,-84.532,167.132,43.146,157.953
C06898=1029.114,-102.060,-84.542,167.134,43.145,157.953
C06899=1029.120,-101.810,-84.551,167.137,43.143,157.953
C06900=1029.126,-101.561,-84.561,167.140,43.141,157.953
C06901=1029.132,-101.311,-84.570,167.143,43.139,157.953
C06902=1029.139,-101.025,-84.581,167.146,43.137,157.953
C06903=1029.145,-100.737,-84.593,167.150,43.134,157.952
C06904=1029.152,-100.451,-84.604,167.153,43.132,157.952
C06905=1029.159,-100.164,-84.615,167.157,43.130,157.952
C06906=1029.165,-99.914,-84.624,167.159,43.128,157.952
C06907=1029.171,-99.664,-84.634,167.162,43.126,157.952
C06908=1029.177,-99.415,-84.643,167.166,43.124,157.952
C06909=1029.182,-99.165,-84.653,167.168,43.122,157.952
C06910=1029.188,-98.916,-84.663,167.171,43.120,157.952
C06911=1029.195,-98.666,-84.673,167.174,43.118,157.951
C06912=1029.201,-98.416,-84.683,167.177,43.116,157.951
C06913=1029.206,-98.166,-84.693,167.180,43.114,157.951
C06914=1029.212,-97.917,-84.702,167.183,43.112,157.951
C06915=1029.219,-97.667,-84.712,167.185,43.110,157.951
C06916=1029.224,-97.417,-84.722,167.189,43.108,157.951
C06917=1029.230,-97.168,-84.731,167.192,43.106,157.951
C06918=1029.235,-96.918,-84.742,167.194,43.104,157.951
C06919=1029.241,-96.668,-84.752,167.197,43.102,157.951
C06920=1029.247,-96.418,-84.762,167.200,43.100,157.950
C06921=1029.253,-96.168,-84.771,167.203,43.098,157.950
C06922=1029.259,-95.919,-84.782,167.206,43.097,157.950
C06923=1029.265,-95.669,-84.792,167.209,43.095,157.950
C06924=1029.270,-95.419,-84.802,167.211,43.093,157.950
C06925=1029.277,-95.169,-84.812,167.214,43.091,157.950
C06926=1029.282,-94.920,-84.822,167.218,43.090,157.950
C06927=1029.288,-94.671,-84.832,167.220,43.088,157.950
C06928=1029.293,-94.420,-84.842,167.223,43.086,157.950
C06929=1029.300,-94.171,-84.852,167.226,43.084,157.950
C06930=1029.305,-93.921,-84.862,167.228,43.082,157.950
C06931=1029.311,-93.671,-84.872,167.232,43.080,157.949
C06932=1029.317,-93.421,-84.882,167.235,43.078,157.949
C06933=1029.323,-93.172,-84.892,167.237,43.077,157.949
C06934=1029.329,-92.922,-84.902,167.240,43.075,157.949
C06935=1029.335,-92.673,-84.913,167.243,43.073,157.949
C06936=1029.341,-92.423,-84.923,167.246,43.071,157.949
C06937=1029.347,-92.173,-84.932,167.249,43.069,157.949
C06938=1029.353,-91.923,-84.943,167.252,43.067,157.949
C06939=1029.359,-91.674,-84.953,167.254,43.065,157.949
C06940=1029.364,-91.423,-84.963,167.257,43.063,157.948
C06941=1029.371,-91.174,-84.973,167.261,43.061,157.948
C06942=1029.376,-90.924,-84.983,167.263,43.060,157.948
C06943=1029.383,-90.675,-84.994,167.266,43.058,157.948
C06944=1029.388,-90.425,-85.004,167.269,43.056,157.948
C06945=1029.394,-90.176,-85.014,167.272,43.055,157.948
C06946=1029.400,-89.926,-85.024,167.275,43.053,157.948
C06947=1029.406,-89.676,-85.034,167.278,43.051,157.948
C06948=1029.412,-89.426,-85.045,167.281,43.049,157.948
C06949=1029.417,-89.176,-85.055,167.283,43.047,157.948
C06950=1029.424,-88.927,-85.065,167.286,43.045,157.948
C06951=1029.430,-88.676,-85.076,167.289,43.043,157.947
C06952=1029.436,-88.427,-85.086,167.292,43.041,157.947
C06953=1029.442,-88.177,-85.096,167.295,43.040,157.947
C06954=1029.448,-87.928,-85.107,167.298,43.038,157.947
C06955=1029.454,-87.678,-85.117,167.300,43.036,157.947
C06956=1029.460,-87.428,-85.127,167.303,43.034,157.947
C06957=1029.466,-87.179,-85.138,167.307,43.032,157.947
C06958=1029.471,-86.929,-85.148,167.309,43.030,157.947
C06959=1029.478,-86.680,-85.158,167.312,43.028,157.947
C06960=1029.483,-86.430,-85.168,167.315,43.026,157.946
C06961=1029.490,-86.180,-85.179,167.317,43.025,157.946
C06962=1029.496,-85.930,-85.189,167.321,43.023,157.946
C06963=1029.502,-85.680,-85.200,167.324,43.021,157.946
C06964=1029.508,-85.431,-85.210,167.326,43.019,157.946
C06965=1029.514,-85.181,-85.220,167.329,43.017,157.946
C06966=1029.521,-84.896,-85.232,167.333,43.015,157.946
C06967=1029.528,-84.612,-85.244,167.335,43.013,157.946
C06968=1029.535,-84.328,-85.256,167.339,43.011,157.946
C06969=1029.541,-84.043,-85.268,167.343,43.009,157.946
C06970=1029.547,-83.793,-85.278,167.345,43.007,157.945
C06971=1029.553,-83.544,-85.289,167.348,43.005,157.945
C06972=1029.560,-83.294,-85.300,167.351,43.004,157.945
C06973=1029.566,-83.044,-85.310,167.354,43.002,157.945
C06974=1029.571,-82.794,-85.321,167.357,43.000,157.945
C06975=1029.578,-82.545,-85.331,167.360,42.998,157.945
C06976=1029.584,-82.296,-85.342,167.362,42.996,157.945
C06977=1029.590,-82.045,-85.352,167.365,42.994,157.945
C06978=1029.596,-81.796,-85.363,167.368,42.992,157.945
C06979=1029.602,-81.546,-85.373,167.371,42.990,157.944
C06980=1029.608,-81.296,-85.383,167.374,42.989,157.944
C06981=1029.614,-81.046,-85.394,167.377,42.987,157.944
C06982=1029.621,-80.797,-85.404,167.379,42.985,157.944
C06983=1029.627,-80.548,-85.415,167.382,42.983,157.944
C06984=1029.632,-80.297,-85.426,167.386,42.981,157.944
C06985=1029.639,-80.048,-85.436,167.388,42.979,157.944
C06986=1029.645,-79.798,-85.447,167.391,42.977,157.944
C06987=1029.651,-79.549,-85.458,167.394,42.976,157.944
C06988=1029.657,-79.298,-85.469,167.397,42.974,157.944
C06989=1029.663,-79.049,-85.480,167.399,42.972,157.943
C06990=1029.669,-78.800,-85.490,167.402,42.971,157.943
C06991=1029.675,-78.550,-85.501,167.406,42.969,157.943
C06992=1029.681,-78.299,-85.512,167.408,42.967,157.943
C06993=1029.687,-78.050,-85.523,167.411,42.966,157.943
C06994=1029.692,-77.800,-85.533,167.414,42.964,157.943
C06995=1029.699,-77.550,-85.545,167.416,42.962,157.943
C06996=1029.705,-77.301,-85.555,167.419,42.960,157.943
C06997=1029.711,-77.052,-85.566,167.422,42.959,157.943
C06998=1029.717,-76.802,-85.577,167.425,42.957,157.943
C06999=1029.723,-76.552,-85.588,167.428,42.955,157.943
C07000=1029.729,-76.302,-85.599,167.431,42.953,157.942
C07001=1029.735,-76.053,-85.610,167.434,42.952,157.942
C07002=1029.741,-75.803,-85.621,167.437,42.950,157.942
C07003=1029.747,-75.553,-85.632,167.439,42.948,157.942
C07004=1029.753,-75.304,-85.642,167.442,42.947,157.942
C07005=1029.759,-75.054,-85.653,167.445,42.945,157.942
C07006=1029.765,-74.804,-85.664,167.447,42.944,157.942
C07007=1029.772,-74.554,-85.676,167.451,42.942,157.942
C07008=1029.777,-74.305,-85.686,167.454,42.940,157.942
C07009=1029.783,-74.055,-85.697,167.456,42.938,157.942
C07010=1029.789,-73.805,-85.709,167.459,42.937,157.942
C07011=1029.795,-73.556,-85.720,167.462,42.935,157.942
C07012=1029.801,-73.307,-85.731,167.465,42.933,157.941
C07013=1029.807,-73.056,-85.743,167.467,42.932,157.941
C07014=1029.812,-72.807,-85.754,167.470,42.930,157.941
C07015=1029.818,-72.557,-85.765,167.473,42.929,157.941
C07016=1029.825,-72.307,-85.776,167.476,42.927,157.941
C07017=1029.831,-72.058,-85.787,167.478,42.925,157.941
///RCONF 1,0,0,1,0,0,0,0,0,0,0,0,0,0,0,0,0,0,0,0,0,0,0,0
C07018=1029.836,-71.809,-85.798,167.481,42.924,157.941
C07019=1029.843,-71.558,-85.810,167.484,42.922,157.941
C07020=1029.848,-71.309,-85.821,167.487,42.921,157.941
C07021=1029.854,-71.059,-85.833,167.489,42.919,157.941
C07022=1029.860,-70.810,-85.844,167.492,42.917,157.941
C07023=1029.866,-70.560,-85.855,167.495,42.916,157.941
C07024=1029.872,-70.310,-85.866,167.499,42.914,157.941
C07025=1029.878,-70.061,-85.878,167.501,42.913,157.941
C07026=1029.884,-69.811,-85.889,167.504,42.911,157.941
C07027=1029.890,-69.561,-85.900,167.507,42.909,157.940
C07028=1029.896,-69.311,-85.912,167.510,42.908,157.940
C07029=1029.902,-69.062,-85.923,167.512,42.906,157.940
C07030=1029.909,-68.779,-85.936,167.515,42.905,157.940
C07031=1029.915,-68.497,-85.949,167.519,42.903,157.940
C07032=1029.922,-68.215,-85.961,167.522,42.901,157.940
C07033=1029.929,-67.932,-85.974,167.525,42.899,157.940
C07034=1029.935,-67.683,-85.986,167.528,42.898,157.940
C07035=1029.941,-67.433,-85.998,167.531,42.896,157.940
C07036=1029.946,-67.183,-86.008,167.533,42.895,157.940
C07037=1029.953,-66.934,-86.020,167.536,42.893,157.940
C07038=1029.959,-66.684,-86.031,167.539,42.892,157.940
C07039=1029.965,-66.435,-86.043,167.542,42.890,157.940
C07040=1029.970,-66.185,-86.055,167.544,42.888,157.939
C07041=1029.977,-65.935,-86.066,167.547,42.887,157.939
C07042=1029.983,-65.686,-86.078,167.550,42.885,157.939
C07043=1029.989,-65.436,-86.089,167.553,42.884,157.939
C07044=1029.995,-65.187,-86.100,167.555,42.882,157.939
C07045=1030.001,-64.936,-86.112,167.558,42.880,157.939
C07046=1030.007,-64.687,-86.124,167.561,42.879,157.939
C07047=1030.013,-64.437,-86.135,167.563,42.877,157.939
C07048=1030.020,-64.187,-86.146,167.566,42.875,157.939
C07049=1030.026,-63.938,-86.158,167.569,42.874,157.939
C07050=1030.031,-63.688,-86.170,167.572,42.872,157.939
C07051=1030.037,-63.439,-86.181,167.575,42.871,157.939
C07052=1030.044,-63.189,-86.193,167.577,42.869,157.939
C07053=1030.050,-62.939,-86.205,167.580,42.867,157.938
C07054=1030.056,-62.690,-86.215,167.583,42.866,157.938
C07055=1030.062,-62.440,-86.228,167.585,42.864,157.938
C07056=1030.068,-62.191,-86.240,167.589,42.862,157.938
C07057=1030.074,-61.941,-86.251,167.592,42.861,157.938
C07058=1030.081,-61.691,-86.263,167.595,42.859,157.938
C07059=1030.086,-61.441,-86.274,167.597,42.858,157.938
C07060=1030.093,-61.192,-86.286,167.600,42.856,157.938
C07061=1030.098,-60.942,-86.297,167.603,42.855,157.938
C07062=1030.105,-60.693,-86.309,167.606,42.854,157.938
C07063=1030.111,-60.442,-86.321,167.608,42.852,157.938
C07064=1030.117,-60.193,-86.332,167.611,42.850,157.938
C07065=1030.123,-59.944,-86.344,167.614,42.849,157.938
C07066=1030.130,-59.694,-86.356,167.617,42.847,157.938
C07067=1030.136,-59.445,-86.367,167.619,42.845,157.937
C07068=1030.142,-59.195,-86.380,167.622,42.844,157.937
C07069=1030.148,-58.945,-86.391,167.625,42.842,157.937
C07070=1030.154,-58.696,-86.403,167.627,42.840,157.937
C07071=1030.161,-58.446,-86.415,167.630,42.839,157.937
C07072=1030.166,-58.196,-86.426,167.633,42.837,157.937
C07073=1030.172,-57.947,-86.438,167.636,42.835,157.937
C07074=1030.179,-57.697,-86.450,167.638,42.834,157.937
C07075=1030.185,-57.447,-86.461,167.641,42.832,157.937
C07076=1030.191,-57.197,-86.474,167.644,42.831,157.937
C07077=1030.197,-56.948,-86.485,167.647,42.829,157.937
C07078=1030.203,-56.698,-86.497,167.649,42.828,157.937
C07079=1030.210,-56.449,-86.509,167.652,42.826,157.936
C07080=1030.216,-56.199,-86.521,167.655,42.825,157.936
C07081=1030.222,-55.950,-86.533,167.657,42.823,157.936
C07082=1030.228,-55.700,-86.544,167.660,42.821,157.936
C07083=1030.234,-55.450,-86.557,167.663,42.820,157.936
C07084=1030.241,-55.200,-86.569,167.666,42.818,157.936
C07085=1030.247,-54.951,-86.580,167.668,42.816,157.936
C07086=1030.253,-54.701,-86.591,167.671,42.815,157.936
C07087=1030.259,-54.451,-86.604,167.674,42.813,157.936
C07088=1030.266,-54.202,-86.616,167.677,42.811,157.936
C07089=1030.272,-53.953,-86.627,167.679,42.810,157.936
C07090=1030.279,-53.703,-86.639,167.682,42.808,157.936
C07091=1030.284,-53.453,-86.651,167.685,42.807,157.935
C07092=1030.291,-53.203,-86.663,167.689,42.805,157.935
C07093=1030.298,-52.954,-86.675,167.691,42.803,157.935
C07094=1030.304,-52.672,-86.689,167.694,42.802,157.935
C07095=1030.311,-52.392,-86.702,167.697,42.800,157.935
C07096=1030.318,-52.110,-86.715,167.700,42.798,157.935
C07097=1030.326,-51.829,-86.729,167.703,42.796,157.935
C07098=1030.332,-51.579,-86.742,167.706,42.795,157.935
C07099=1030.338,-51.331,-86.753,167.708,42.793,157.935
C07100=1030.345,-51.081,-86.765,167.711,42.791,157.935
C07101=1030.350,-50.831,-86.777,167.714,42.790,157.935
C07102=1030.357,-50.581,-86.789,167.717,42.788,157.934
C07103=1030.363,-50.331,-86.802,167.720,42.787,157.935
C07104=1030.369,-50.081,-86.814,167.722,42.785,157.934
C07105=1030.375,-49.832,-86.826,167.725,42.784,157.934
C07106=1030.381,-49.582,-86.839,167.728,42.782,157.934
C07107=1030.387,-49.333,-86.850,167.731,42.781,157.934
C07108=1030.393,-49.083,-86.863,167.733,42.780,157.934
C07109=1030.399,-48.834,-86.876,167.736,42.778,157.934
C07110=1030.406,-48.584,-86.888,167.739,42.777,157.934
C07111=1030.412,-48.334,-86.901,167.742,42.775,157.934
C07112=1030.418,-48.084,-86.913,167.743,42.774,157.934
C07113=1030.424,-47.836,-86.925,167.746,42.772,157.934
C07114=1030.430,-47.586,-86.937,167.749,42.771,157.934
///RCONF 1,0,0,0,0,0,0,0,0,0,0,0,0,0,0,0,0,0,0,0,0,0,0,0
C07115=1030.436,-47.336,-86.950,167.752,42.769,157.934
C07116=1030.442,-47.086,-86.962,167.755,42.768,157.934
C07117=1030.448,-46.836,-86.974,167.757,42.767,157.934
C07118=1030.454,-46.587,-86.988,167.760,42.765,157.934
C07119=1030.461,-46.337,-87.000,167.763,42.764,157.934
C07120=1030.467,-46.088,-87.012,167.766,42.762,157.933
C07121=1030.473,-45.838,-87.025,167.768,42.761,157.933
C07122=1030.480,-45.588,-87.037,167.771,42.759,157.933
C07123=1030.485,-45.340,-87.050,167.774,42.758,157.933
C07124=1030.491,-45.090,-87.062,167.776,42.757,157.933
C07125=1030.498,-44.840,-87.074,167.779,42.755,157.933
C07126=1030.504,-44.590,-87.087,167.781,42.754,157.933
C07127=1030.510,-44.340,-87.099,167.784,42.752,157.933
C07128=1030.517,-44.091,-87.112,167.787,42.751,157.933
C07129=1030.522,-43.841,-87.124,167.790,42.750,157.933
C07130=1030.528,-43.592,-87.137,167.792,42.748,157.933
C07131=1030.534,-43.342,-87.150,167.795,42.747,157.933
C07132=1030.541,-43.093,-87.162,167.798,42.745,157.933
C07133=1030.547,-42.843,-87.175,167.801,42.744,157.933
C07134=1030.553,-42.593,-87.187,167.803,42.742,157.933
C07135=1030.560,-42.343,-87.199,167.806,42.741,157.933
C07136=1030.566,-42.094,-87.213,167.808,42.740,157.932
C07137=1030.572,-41.844,-87.225,167.811,42.738,157.932
C07138=1030.578,-41.595,-87.237,167.814,42.737,157.932
C07139=1030.585,-41.345,-87.250,167.816,42.735,157.932
C07140=1030.591,-41.096,-87.263,167.819,42.734,157.932
C07141=1030.596,-40.846,-87.275,167.822,42.732,157.932
C07142=1030.603,-40.597,-87.288,167.825,42.731,157.932
C07143=1030.609,-40.347,-87.301,167.827,42.729,157.932
C07144=1030.615,-40.097,-87.313,167.830,42.728,157.932
C07145=1030.622,-39.848,-87.326,167.833,42.727,157.932
C07146=1030.628,-39.598,-87.338,167.836,42.725,157.932
C07147=1030.634,-39.349,-87.352,167.837,42.724,157.932
C07148=1030.640,-39.099,-87.364,167.840,42.722,157.932
C07149=1030.647,-38.849,-87.376,167.843,42.721,157.932
C07150=1030.653,-38.600,-87.390,167.846,42.719,157.932
C07151=1030.660,-38.350,-87.402,167.849,42.718,157.932
C07152=1030.666,-38.100,-87.416,167.851,42.717,157.932
C07153=1030.672,-37.850,-87.428,167.854,42.715,157.931
C07154=1030.678,-37.601,-87.442,167.856,42.714,157.931
C07155=1030.684,-37.351,-87.454,167.859,42.713,157.931
C07156=1030.690,-37.102,-87.467,167.861,42.711,157.931
C07157=1030.696,-36.852,-87.480,167.864,42.710,157.931
C07158=1030.703,-36.572,-87.495,167.867,42.709,157.931
C07159=1030.710,-36.291,-87.509,167.870,42.707,157.931
C07160=1030.717,-36.010,-87.524,167.874,42.706,157.931
C07161=1030.723,-35.730,-87.539,167.876,42.704,157.931
C07162=1030.730,-35.480,-87.552,167.879,42.703,157.931
C07163=1030.736,-35.230,-87.564,167.881,42.701,157.931
C07164=1030.742,-34.981,-87.578,167.884,42.700,157.931
C07165=1030.748,-34.732,-87.591,167.887,42.699,157.931
C07166=1030.754,-34.482,-87.603,167.889,42.697,157.931
C07167=1030.761,-34.232,-87.617,167.892,42.696,157.931
C07168=1030.767,-33.982,-87.630,167.895,42.695,157.931
C07169=1030.773,-33.733,-87.643,167.897,42.693,157.930
C07170=1030.779,-33.484,-87.656,167.899,42.692,157.930
C07171=1030.785,-33.234,-87.669,167.902,42.691,157.930
C07172=1030.791,-32.984,-87.682,167.905,42.689,157.930
C07173=1030.797,-32.735,-87.695,167.908,42.688,157.930
C07174=1030.804,-32.485,-87.708,167.911,42.686,157.930
C07175=1030.810,-32.235,-87.721,167.912,42.685,157.930
C07176=1030.816,-31.986,-87.735,167.915,42.684,157.930
C07177=1030.822,-31.736,-87.747,167.918,42.682,157.930
C07178=1030.829,-31.487,-87.760,167.921,42.681,157.930
C07179=1030.835,-31.238,-87.773,167.924,42.680,157.930
C07180=1030.842,-30.988,-87.787,167.926,42.678,157.930
C07181=1030.847,-30.738,-87.800,167.928,42.677,157.930
C07182=1030.854,-30.489,-87.813,167.931,42.675,157.930
C07183=1030.860,-30.239,-87.827,167.934,42.674,157.930
C07184=1030.867,-29.989,-87.840,167.937,42.673,157.930
C07185=1030.873,-29.739,-87.853,167.939,42.671,157.930
C07186=1030.879,-29.490,-87.866,167.942,42.670,157.930
C07187=1030.885,-29.241,-87.879,167.944,42.669,157.930
C07188=1030.891,-28.992,-87.893,167.947,42.667,157.929
C07189=1030.898,-28.741,-87.905,167.949,42.666,157.929
C07190=1030.904,-28.492,-87.919,167.952,42.664,157.929
C07191=1030.910,-28.243,-87.932,167.955,42.663,157.929
C07192=1030.916,-27.993,-87.945,167.958,42.662,157.929
C07193=1030.923,-27.743,-87.959,167.959,42.660,157.929
C07194=1030.929,-27.493,-87.971,167.962,42.659,157.929
C07195=1030.935,-27.244,-87.985,167.965,42.657,157.929
C07196=1030.942,-26.994,-87.998,167.968,42.656,157.929
C07197=1030.948,-26.745,-88.012,167.971,42.655,157.929
C07198=1030.954,-26.495,-88.026,167.973,42.654,157.929
C07199=1030.960,-26.246,-88.039,167.975,42.652,157.929
C07200=1030.967,-25.996,-88.052,167.978,42.651,157.929
C07201=1030.973,-25.747,-88.066,167.981,42.650,157.929
C07202=1030.979,-25.497,-88.080,167.983,42.649,157.929
C07203=1030.985,-25.248,-88.093,167.986,42.648,157.929
C07204=1030.992,-24.998,-88.106,167.988,42.646,157.929
C07205=1030.998,-24.749,-88.120,167.991,42.645,157.929
C07206=1031.003,-24.499,-88.134,167.993,42.644,157.929
C07207=1031.010,-24.249,-88.147,167.996,42.643,157.929
C07208=1031.016,-24.000,-88.161,167.999,42.641,157.928
